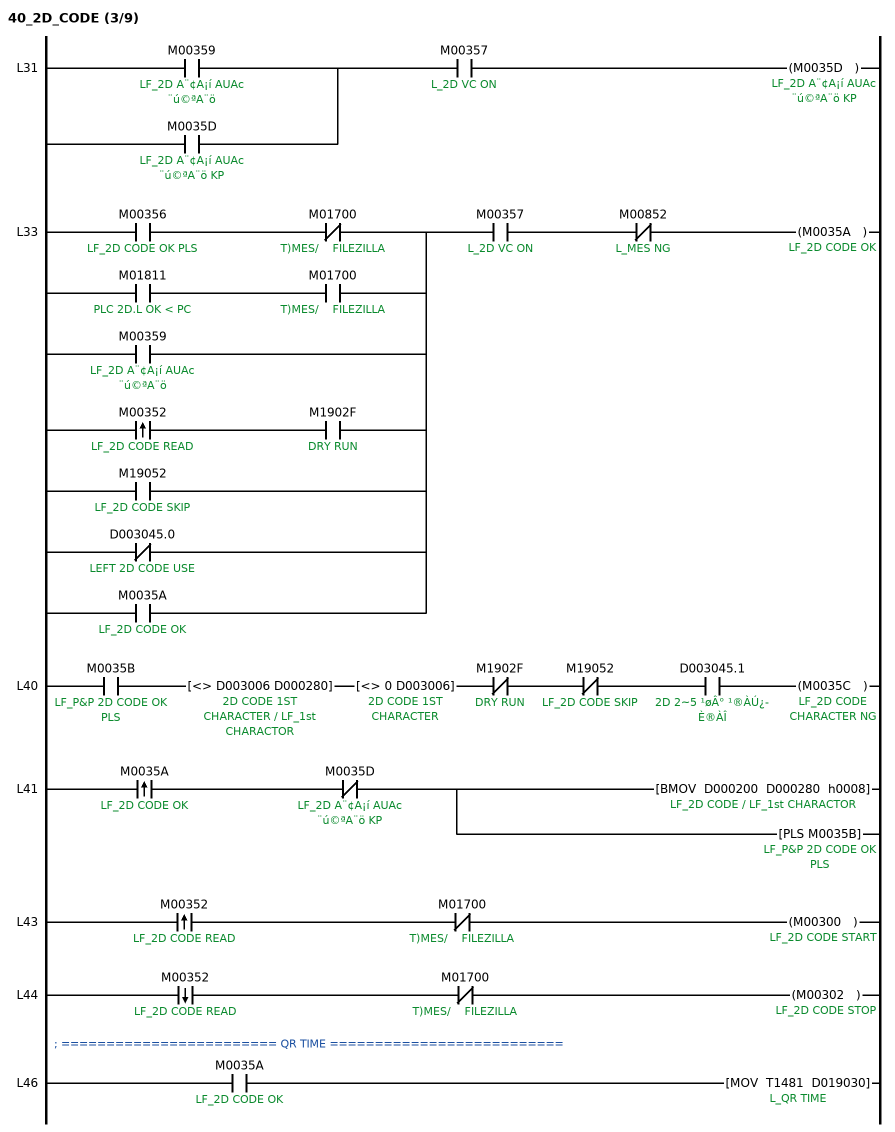
[picture p240: 40_2D_CODE rungs L31-L46]
; L31
LOAD      M00359	// LF_2D A¨¢A¡í AUAc ¨ú©ªA¨ö
OR        M0035D	// LF_2D A¨¢A¡í AUAc ¨ú©ªA¨ö KP
AND       M00357	// L_2D VC ON
OUT       M0035D	// LF_2D A¨¢A¡í AUAc ¨ú©ªA¨ö KP
; L33
LOAD      M00356	// LF_2D CODE OK PLS
AND NOT   M01700	// T)MES/    FILEZILLA
LOAD      M01811	// PLC 2D.L OK < PC
AND       M01700	// T)MES/    FILEZILLA
OR LOAD
OR        M00359	// LF_2D A¨¢A¡í AUAc ¨ú©ªA¨ö
LOADP     M00352	// LF_2D CODE READ
AND       M1902F	// DRY RUN
OR LOAD
OR        M19052	// LF_2D CODE SKIP
OR NOT    D003045.0	// LEFT 2D CODE USE
OR        M0035A	// LF_2D CODE OK
AND       M00357	// L_2D VC ON
AND NOT   M00852	// L_MES NG
OUT       M0035A	// LF_2D CODE OK
; L40
LOAD      M0035B	// LF_P&P 2D CODE OK PLS
AND<>     D003006 D000280	// 2D CODE 1ST CHARACTER / LF_1st CHARACTOR
AND<>     0 D003006	// 2D CODE 1ST CHARACTER
AND NOT   M1902F	// DRY RUN
AND NOT   M19052	// LF_2D CODE SKIP
AND       D003045.1	// 2D 2~5 ¹øÂ° ¹®ÀÚ¿­ È®ÀÎ
OUT       M0035C	// LF_2D CODE CHARACTER NG
; L41
LOADP     M0035A	// LF_2D CODE OK
AND NOT   M0035D	// LF_2D A¨¢A¡í AUAc ¨ú©ªA¨ö KP
BMOV      D000200 D000280 h0008	// LF_2D CODE / LF_1st CHARACTOR
OUTP      M0035B	// LF_P&P 2D CODE OK PLS
; L43
LOADP     M00352	// LF_2D CODE READ
AND NOT   M01700	// T)MES/    FILEZILLA
OUT       M00300	// LF_2D CODE START
; L44
LOADN     M00352	// LF_2D CODE READ
AND NOT   M01700	// T)MES/    FILEZILLA
OUT       M00302	// LF_2D CODE STOP
// ======================== QR TIME ==========================
; L46
LOAD      M0035A	// LF_2D CODE OK
MOV       T1481 D019030	// L_QR TIME

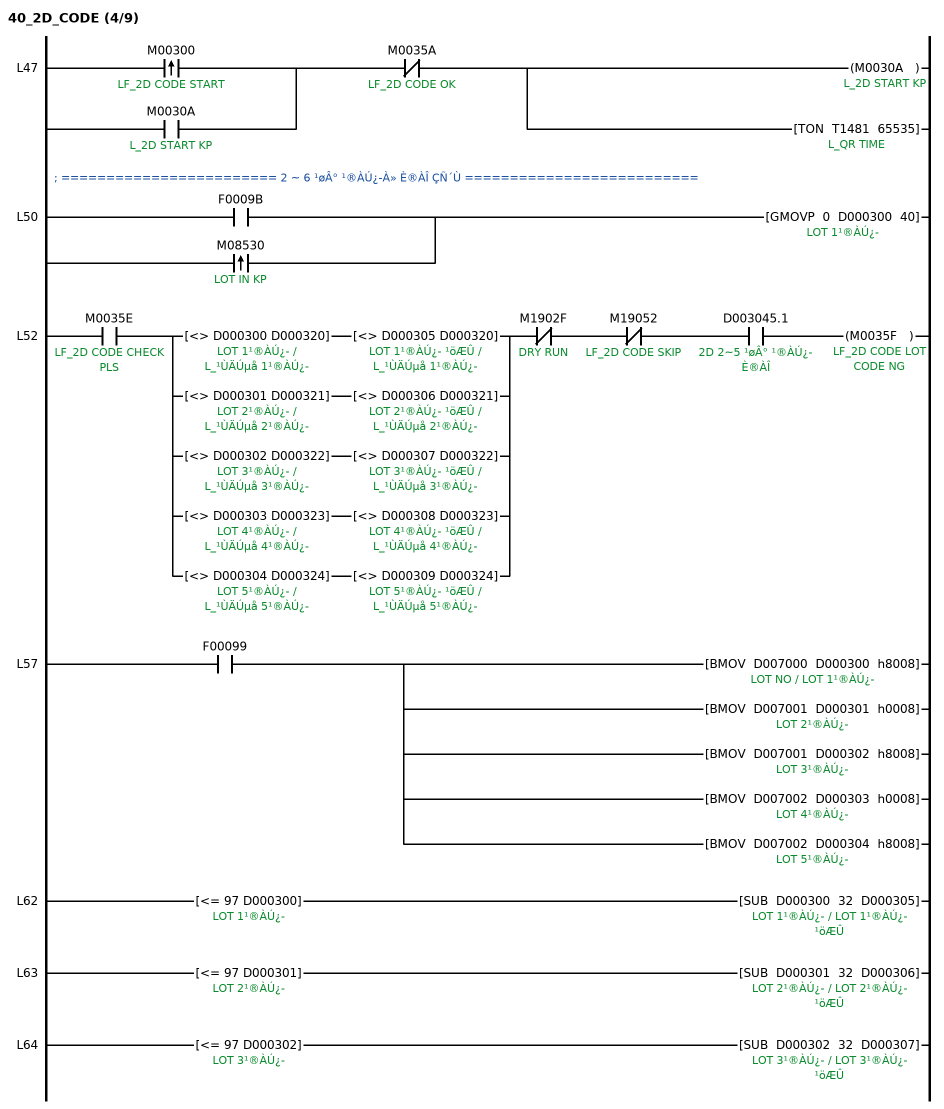
; L47
LOADP     M00300	// LF_2D CODE START
OR        M0030A	// L_2D START KP
AND NOT   M0035A	// LF_2D CODE OK
OUT       M0030A	// L_2D START KP
TON       T1481 65535	// L_QR TIME
// ======================== 2 ~ 6 ¹øÂ° ¹®ÀÚ¿­À» È®ÀÎ ÇÑ´Ù ==========================
; L50
LOAD      F0009B
ORP       M08530	// LOT IN KP
GMOVP     0 D000300 40	// LOT 1¹®ÀÚ¿­
; L52
LOAD      M0035E	// LF_2D CODE CHECK PLS
LOAD<>    D000300 D000320	// LOT 1¹®ÀÚ¿­ / L_¹ÙÄÚµå 1¹®ÀÚ¿­
AND<>     D000305 D000320	// LOT 1¹®ÀÚ¿­ ¹öÆÛ / L_¹ÙÄÚµå 1¹®ÀÚ¿­
LOAD<>    D000301 D000321	// LOT 2¹®ÀÚ¿­ / L_¹ÙÄÚµå 2¹®ÀÚ¿­
AND<>     D000306 D000321	// LOT 2¹®ÀÚ¿­ ¹öÆÛ / L_¹ÙÄÚµå 2¹®ÀÚ¿­
OR LOAD
LOAD<>    D000302 D000322	// LOT 3¹®ÀÚ¿­ / L_¹ÙÄÚµå 3¹®ÀÚ¿­
AND<>     D000307 D000322	// LOT 3¹®ÀÚ¿­ ¹öÆÛ / L_¹ÙÄÚµå 3¹®ÀÚ¿­
OR LOAD
LOAD<>    D000303 D000323	// LOT 4¹®ÀÚ¿­ / L_¹ÙÄÚµå 4¹®ÀÚ¿­
AND<>     D000308 D000323	// LOT 4¹®ÀÚ¿­ ¹öÆÛ / L_¹ÙÄÚµå 4¹®ÀÚ¿­
OR LOAD
LOAD<>    D000304 D000324	// LOT 5¹®ÀÚ¿­ / L_¹ÙÄÚµå 5¹®ÀÚ¿­
AND<>     D000309 D000324	// LOT 5¹®ÀÚ¿­ ¹öÆÛ / L_¹ÙÄÚµå 5¹®ÀÚ¿­
OR LOAD
AND LOAD
AND NOT   M1902F	// DRY RUN
AND NOT   M19052	// LF_2D CODE SKIP
AND       D003045.1	// 2D 2~5 ¹øÂ° ¹®ÀÚ¿­ È®ÀÎ
OUT       M0035F	// LF_2D CODE LOT CODE NG
; L57
LOAD      F00099
BMOV      D007000 D000300 h8008	// LOT NO / LOT 1¹®ÀÚ¿­
BMOV      D007001 D000301 h0008	// LOT 2¹®ÀÚ¿­
BMOV      D007001 D000302 h8008	// LOT 3¹®ÀÚ¿­
BMOV      D007002 D000303 h0008	// LOT 4¹®ÀÚ¿­
BMOV      D007002 D000304 h8008	// LOT 5¹®ÀÚ¿­
; L62
LOAD<=    97 D000300	// LOT 1¹®ÀÚ¿­
SUB       D000300 32 D000305	// LOT 1¹®ÀÚ¿­ / LOT 1¹®ÀÚ¿­ ¹öÆÛ
; L63
LOAD<=    97 D000301	// LOT 2¹®ÀÚ¿­
SUB       D000301 32 D000306	// LOT 2¹®ÀÚ¿­ / LOT 2¹®ÀÚ¿­ ¹öÆÛ
; L64
LOAD<=    97 D000302	// LOT 3¹®ÀÚ¿­
SUB       D000302 32 D000307	// LOT 3¹®ÀÚ¿­ / LOT 3¹®ÀÚ¿­ ¹öÆÛ

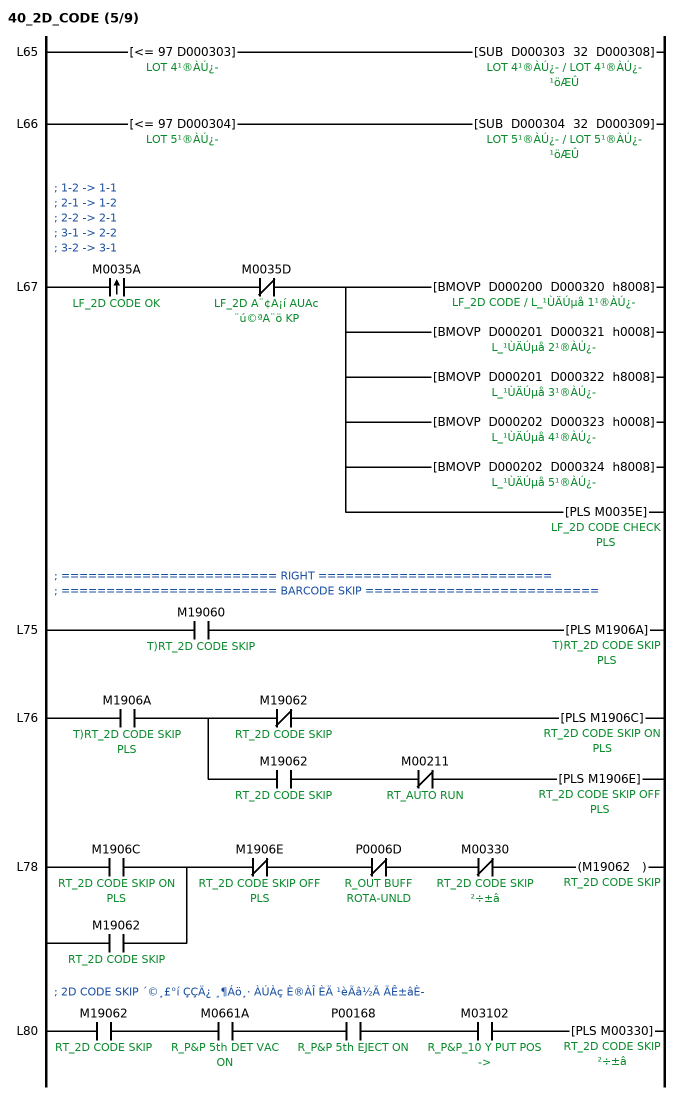
; L65
LOAD<=    97 D000303	// LOT 4¹®ÀÚ¿­
SUB       D000303 32 D000308	// LOT 4¹®ÀÚ¿­ / LOT 4¹®ÀÚ¿­ ¹öÆÛ
; L66
LOAD<=    97 D000304	// LOT 5¹®ÀÚ¿­
SUB       D000304 32 D000309	// LOT 5¹®ÀÚ¿­ / LOT 5¹®ÀÚ¿­ ¹öÆÛ
; L67
LOADP     M0035A	// LF_2D CODE OK
AND NOT   M0035D	// LF_2D A¨¢A¡í AUAc ¨ú©ªA¨ö KP
BMOVP     D000200 D000320 h8008	// LF_2D CODE / L_¹ÙÄÚµå 1¹®ÀÚ¿­
BMOVP     D000201 D000321 h0008	// L_¹ÙÄÚµå 2¹®ÀÚ¿­
BMOVP     D000201 D000322 h8008	// L_¹ÙÄÚµå 3¹®ÀÚ¿­
BMOVP     D000202 D000323 h0008	// L_¹ÙÄÚµå 4¹®ÀÚ¿­
BMOVP     D000202 D000324 h8008	// L_¹ÙÄÚµå 5¹®ÀÚ¿­
OUTP      M0035E	// LF_2D CODE CHECK PLS
// output comment: 1-2 -> 1-1
// output comment: 2-1 -> 1-2
// output comment: 2-2 -> 2-1
// output comment: 3-1 -> 2-2
// output comment: 3-2 -> 3-1
// ======================== RIGHT ==========================
// ======================== BARCODE SKIP ==========================
; L75
LOAD      M19060	// T)RT_2D CODE SKIP
OUTP      M1906A	// T)RT_2D CODE SKIP PLS
; L76
LOAD      M1906A	// T)RT_2D CODE SKIP PLS
MPUSH
AND NOT   M19062	// RT_2D CODE SKIP
OUTP      M1906C	// RT_2D CODE SKIP ON PLS
MPOP
AND       M19062	// RT_2D CODE SKIP
AND NOT   M00211	// RT_AUTO RUN
OUTP      M1906E	// RT_2D CODE SKIP OFF PLS
; L78
LOAD      M1906C	// RT_2D CODE SKIP ON PLS
OR        M19062	// RT_2D CODE SKIP
AND NOT   M1906E	// RT_2D CODE SKIP OFF PLS
AND NOT   P0006D	// R_OUT BUFF ROTA-UNLD
AND NOT   M00330	// RT_2D CODE SKIP ²÷±â
OUT       M19062	// RT_2D CODE SKIP
; L80
LOAD      M19062	// RT_2D CODE SKIP
AND       M0661A	// R_P&P 5th DET VAC ON
AND       P00168	// R_P&P 5th EJECT ON
AND       M03102	// R_P&P_10 Y PUT POS ->
OUTP      M00330	// RT_2D CODE SKIP ²÷±â
// output comment: 2D CODE SKIP ´©¸£°í ÇÇÄ¿ ¸¶Áö¸· ÀÚÀç È®ÀÎ ÈÄ ¹èÃâ½Ã ÃÊ±âÈ­

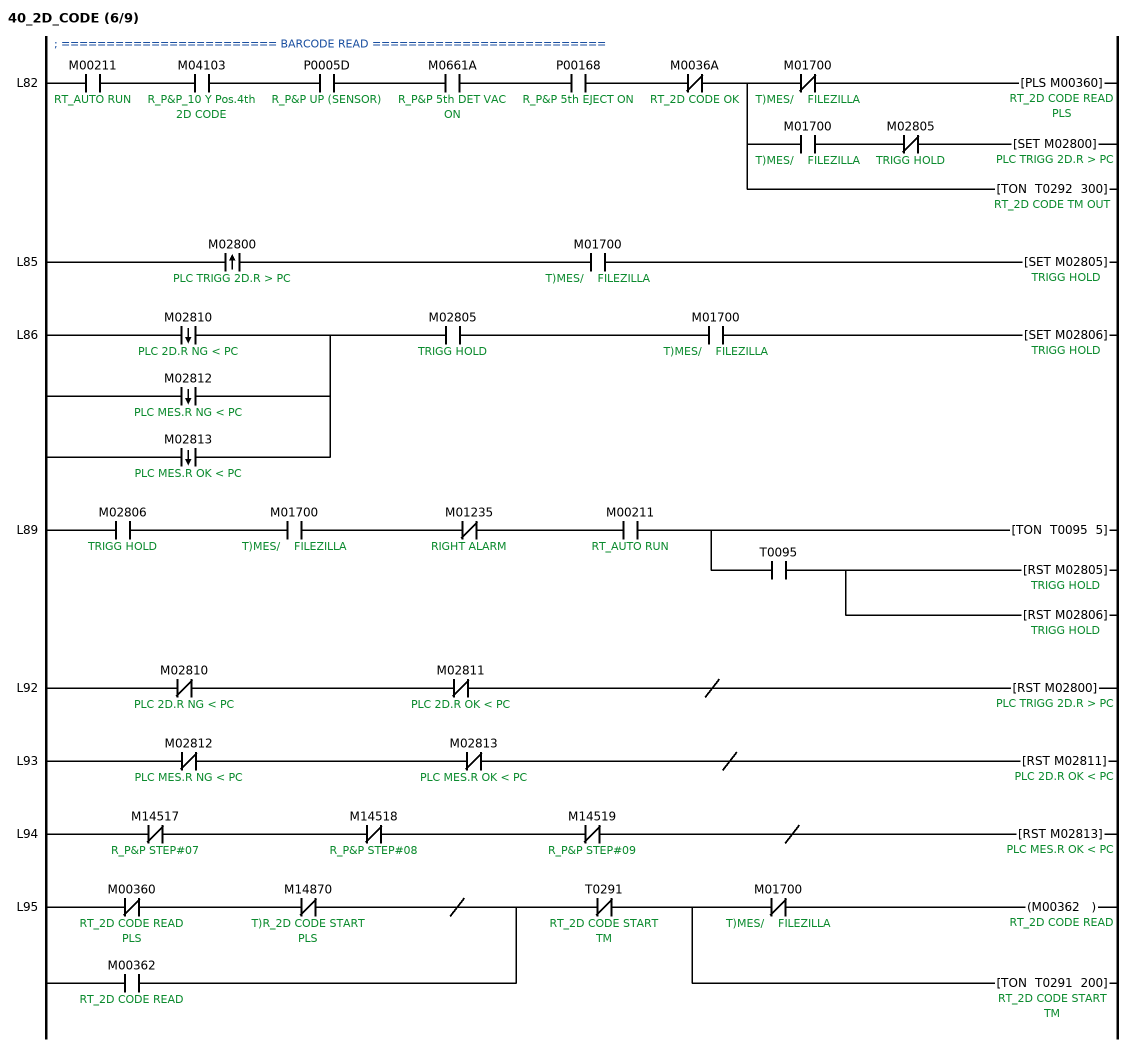
// ======================== BARCODE READ ==========================
; L82
LOAD      M00211	// RT_AUTO RUN
AND       M04103	// R_P&P_10 Y Pos.4th 2D CODE
AND       P0005D	// R_P&P UP (SENSOR)
AND       M0661A	// R_P&P 5th DET VAC ON
AND       P00168	// R_P&P 5th EJECT ON
AND NOT   M0036A	// RT_2D CODE OK
MPUSH
AND NOT   M01700	// T)MES/    FILEZILLA
OUTP      M00360	// RT_2D CODE READ PLS
MLOAD
AND       M01700	// T)MES/    FILEZILLA
AND NOT   M02805	// TRIGG HOLD
SET       M02800	// PLC TRIGG 2D.R > PC
MPOP
TON       T0292 300	// RT_2D CODE TM OUT
; L85
LOADP     M02800	// PLC TRIGG 2D.R > PC
AND       M01700	// T)MES/    FILEZILLA
SET       M02805	// TRIGG HOLD
; L86
LOADN     M02810	// PLC 2D.R NG < PC
ORN       M02812	// PLC MES.R NG < PC
ORN       M02813	// PLC MES.R OK < PC
AND       M02805	// TRIGG HOLD
AND       M01700	// T)MES/    FILEZILLA
SET       M02806	// TRIGG HOLD
; L89
LOAD      M02806	// TRIGG HOLD
AND       M01700	// T)MES/    FILEZILLA
AND NOT   M01235	// RIGHT ALARM
AND       M00211	// RT_AUTO RUN
TON       T0095 5
AND       T0095
RST       M02805	// TRIGG HOLD
RST       M02806	// TRIGG HOLD
; L92
LOAD NOT  M02810	// PLC 2D.R NG < PC
AND NOT   M02811	// PLC 2D.R OK < PC
NOT
RST       M02800	// PLC TRIGG 2D.R > PC
; L93
LOAD NOT  M02812	// PLC MES.R NG < PC
AND NOT   M02813	// PLC MES.R OK < PC
NOT
RST       M02811	// PLC 2D.R OK < PC
; L94
LOAD NOT  M14517	// R_P&P STEP#07
AND NOT   M14518	// R_P&P STEP#08
AND NOT   M14519	// R_P&P STEP#09
NOT
RST       M02813	// PLC MES.R OK < PC
; L95
LOAD NOT  M00360	// RT_2D CODE READ PLS
AND NOT   M14870	// T)R_2D CODE START PLS
NOT
OR        M00362	// RT_2D CODE READ
AND NOT   T0291	// RT_2D CODE START TM
MPUSH
AND NOT   M01700	// T)MES/    FILEZILLA
OUT       M00362	// RT_2D CODE READ
MPOP
TON       T0291 200	// RT_2D CODE START TM

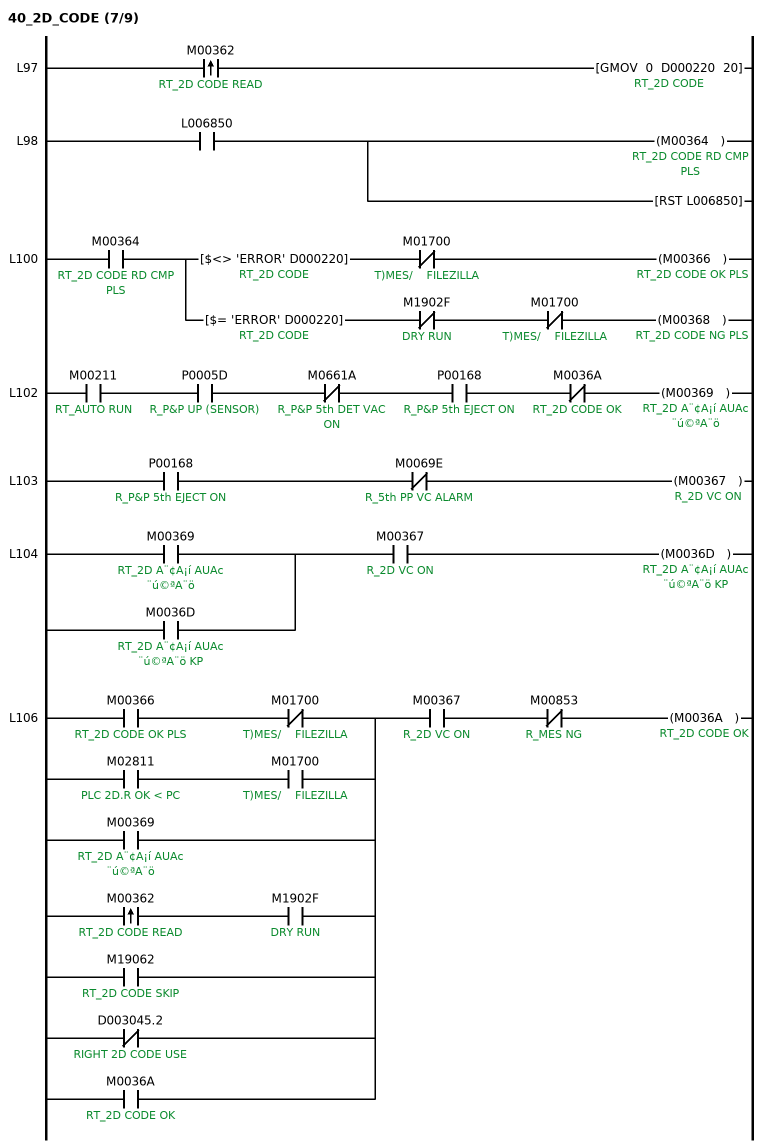
; L97
LOADP     M00362	// RT_2D CODE READ
GMOV      0 D000220 20	// RT_2D CODE
; L98
LOAD      L006850
OUT       M00364	// RT_2D CODE RD CMP PLS
RST       L006850
; L100
LOAD      M00364	// RT_2D CODE RD CMP PLS
MPUSH
AND$<>    'ERROR' D000220	// RT_2D CODE
AND NOT   M01700	// T)MES/    FILEZILLA
OUT       M00366	// RT_2D CODE OK PLS
MPOP
AND$=     'ERROR' D000220	// RT_2D CODE
AND NOT   M1902F	// DRY RUN
AND NOT   M01700	// T)MES/    FILEZILLA
OUT       M00368	// RT_2D CODE NG PLS
; L102
LOAD      M00211	// RT_AUTO RUN
AND       P0005D	// R_P&P UP (SENSOR)
AND NOT   M0661A	// R_P&P 5th DET VAC ON
AND       P00168	// R_P&P 5th EJECT ON
AND NOT   M0036A	// RT_2D CODE OK
OUT       M00369	// RT_2D A¨¢A¡í AUAc ¨ú©ªA¨ö
; L103
LOAD      P00168	// R_P&P 5th EJECT ON
AND NOT   M0069E	// R_5th PP VC ALARM
OUT       M00367	// R_2D VC ON
; L104
LOAD      M00369	// RT_2D A¨¢A¡í AUAc ¨ú©ªA¨ö
OR        M0036D	// RT_2D A¨¢A¡í AUAc ¨ú©ªA¨ö KP
AND       M00367	// R_2D VC ON
OUT       M0036D	// RT_2D A¨¢A¡í AUAc ¨ú©ªA¨ö KP
; L106
LOAD      M00366	// RT_2D CODE OK PLS
AND NOT   M01700	// T)MES/    FILEZILLA
LOAD      M02811	// PLC 2D.R OK < PC
AND       M01700	// T)MES/    FILEZILLA
OR LOAD
OR        M00369	// RT_2D A¨¢A¡í AUAc ¨ú©ªA¨ö
LOADP     M00362	// RT_2D CODE READ
AND       M1902F	// DRY RUN
OR LOAD
OR        M19062	// RT_2D CODE SKIP
OR NOT    D003045.2	// RIGHT 2D CODE USE
OR        M0036A	// RT_2D CODE OK
AND       M00367	// R_2D VC ON
AND NOT   M00853	// R_MES NG
OUT       M0036A	// RT_2D CODE OK

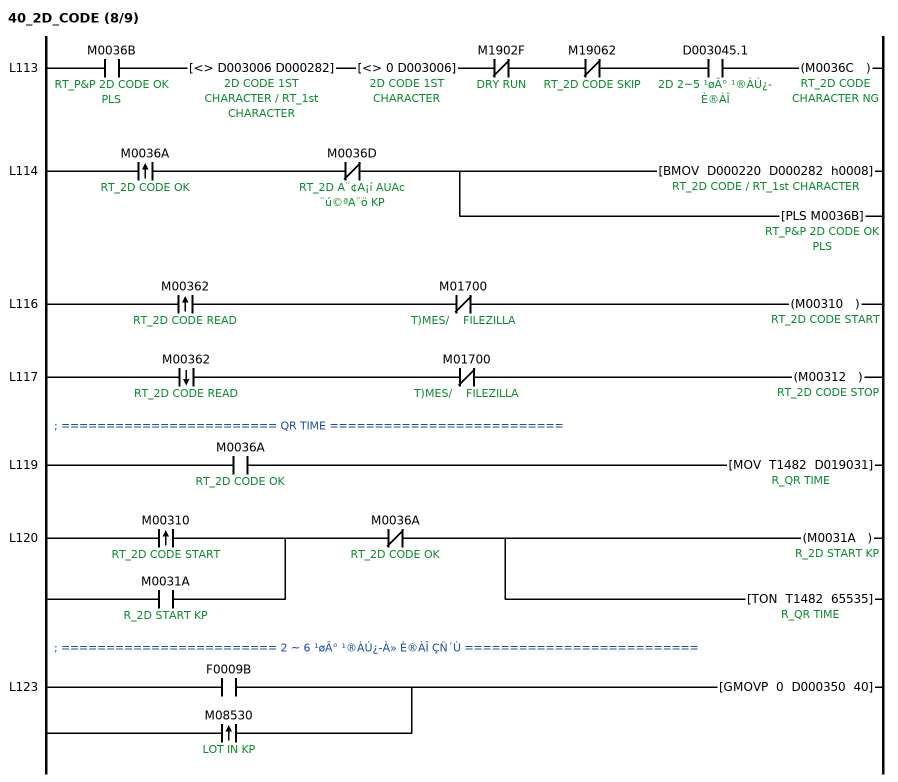
; L113
LOAD      M0036B	// RT_P&P 2D CODE OK PLS
AND<>     D003006 D000282	// 2D CODE 1ST CHARACTER / RT_1st CHARACTER
AND<>     0 D003006	// 2D CODE 1ST CHARACTER
AND NOT   M1902F	// DRY RUN
AND NOT   M19062	// RT_2D CODE SKIP
AND       D003045.1	// 2D 2~5 ¹øÂ° ¹®ÀÚ¿­ È®ÀÎ
OUT       M0036C	// RT_2D CODE CHARACTER NG
; L114
LOADP     M0036A	// RT_2D CODE OK
AND NOT   M0036D	// RT_2D A¨¢A¡í AUAc ¨ú©ªA¨ö KP
BMOV      D000220 D000282 h0008	// RT_2D CODE / RT_1st CHARACTER
OUTP      M0036B	// RT_P&P 2D CODE OK PLS
; L116
LOADP     M00362	// RT_2D CODE READ
AND NOT   M01700	// T)MES/    FILEZILLA
OUT       M00310	// RT_2D CODE START
; L117
LOADN     M00362	// RT_2D CODE READ
AND NOT   M01700	// T)MES/    FILEZILLA
OUT       M00312	// RT_2D CODE STOP
// ======================== QR TIME ==========================
; L119
LOAD      M0036A	// RT_2D CODE OK
MOV       T1482 D019031	// R_QR TIME
; L120
LOADP     M00310	// RT_2D CODE START
OR        M0031A	// R_2D START KP
AND NOT   M0036A	// RT_2D CODE OK
OUT       M0031A	// R_2D START KP
TON       T1482 65535	// R_QR TIME
// ======================== 2 ~ 6 ¹øÂ° ¹®ÀÚ¿­À» È®ÀÎ ÇÑ´Ù ==========================
; L123
LOAD      F0009B
ORP       M08530	// LOT IN KP
GMOVP     0 D000350 40

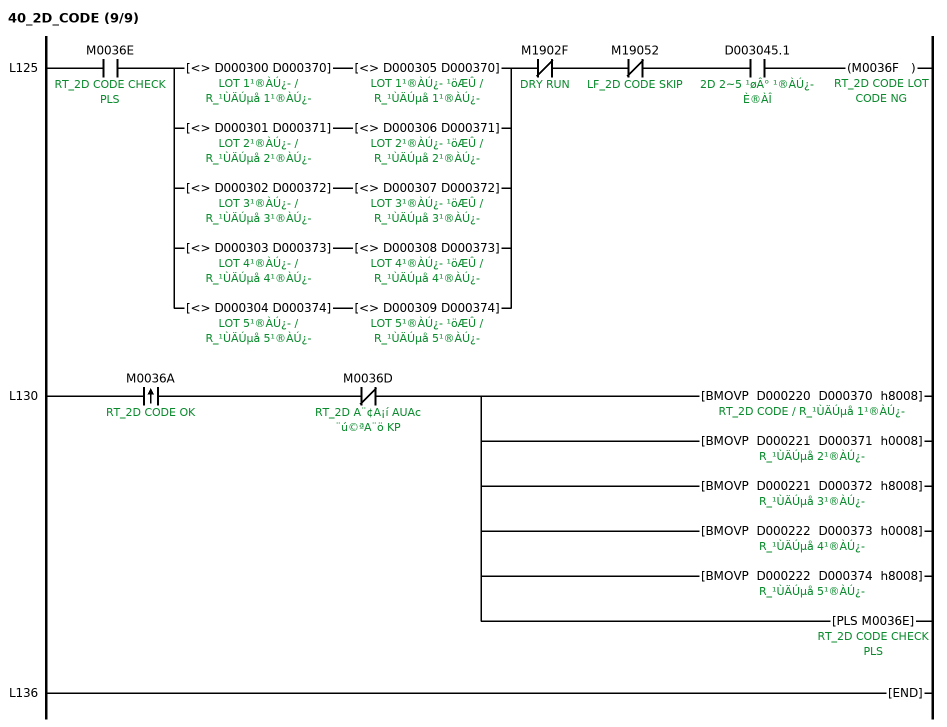
; L125
LOAD      M0036E	// RT_2D CODE CHECK PLS
LOAD<>    D000300 D000370	// LOT 1¹®ÀÚ¿­ / R_¹ÙÄÚµå 1¹®ÀÚ¿­
AND<>     D000305 D000370	// LOT 1¹®ÀÚ¿­ ¹öÆÛ / R_¹ÙÄÚµå 1¹®ÀÚ¿­
LOAD<>    D000301 D000371	// LOT 2¹®ÀÚ¿­ / R_¹ÙÄÚµå 2¹®ÀÚ¿­
AND<>     D000306 D000371	// LOT 2¹®ÀÚ¿­ ¹öÆÛ / R_¹ÙÄÚµå 2¹®ÀÚ¿­
OR LOAD
LOAD<>    D000302 D000372	// LOT 3¹®ÀÚ¿­ / R_¹ÙÄÚµå 3¹®ÀÚ¿­
AND<>     D000307 D000372	// LOT 3¹®ÀÚ¿­ ¹öÆÛ / R_¹ÙÄÚµå 3¹®ÀÚ¿­
OR LOAD
LOAD<>    D000303 D000373	// LOT 4¹®ÀÚ¿­ / R_¹ÙÄÚµå 4¹®ÀÚ¿­
AND<>     D000308 D000373	// LOT 4¹®ÀÚ¿­ ¹öÆÛ / R_¹ÙÄÚµå 4¹®ÀÚ¿­
OR LOAD
LOAD<>    D000304 D000374	// LOT 5¹®ÀÚ¿­ / R_¹ÙÄÚµå 5¹®ÀÚ¿­
AND<>     D000309 D000374	// LOT 5¹®ÀÚ¿­ ¹öÆÛ / R_¹ÙÄÚµå 5¹®ÀÚ¿­
OR LOAD
AND LOAD
AND NOT   M1902F	// DRY RUN
AND NOT   M19052	// LF_2D CODE SKIP
AND       D003045.1	// 2D 2~5 ¹øÂ° ¹®ÀÚ¿­ È®ÀÎ
OUT       M0036F	// RT_2D CODE LOT CODE NG
; L130
LOADP     M0036A	// RT_2D CODE OK
AND NOT   M0036D	// RT_2D A¨¢A¡í AUAc ¨ú©ªA¨ö KP
BMOVP     D000220 D000370 h8008	// RT_2D CODE / R_¹ÙÄÚµå 1¹®ÀÚ¿­
BMOVP     D000221 D000371 h0008	// R_¹ÙÄÚµå 2¹®ÀÚ¿­
BMOVP     D000221 D000372 h8008	// R_¹ÙÄÚµå 3¹®ÀÚ¿­
BMOVP     D000222 D000373 h0008	// R_¹ÙÄÚµå 4¹®ÀÚ¿­
BMOVP     D000222 D000374 h8008	// R_¹ÙÄÚµå 5¹®ÀÚ¿­
OUTP      M0036E	// RT_2D CODE CHECK PLS
; L136
END

PROGRAM 41_MES (task: ½ºÄµ ÇÁ·Î±×·¥)

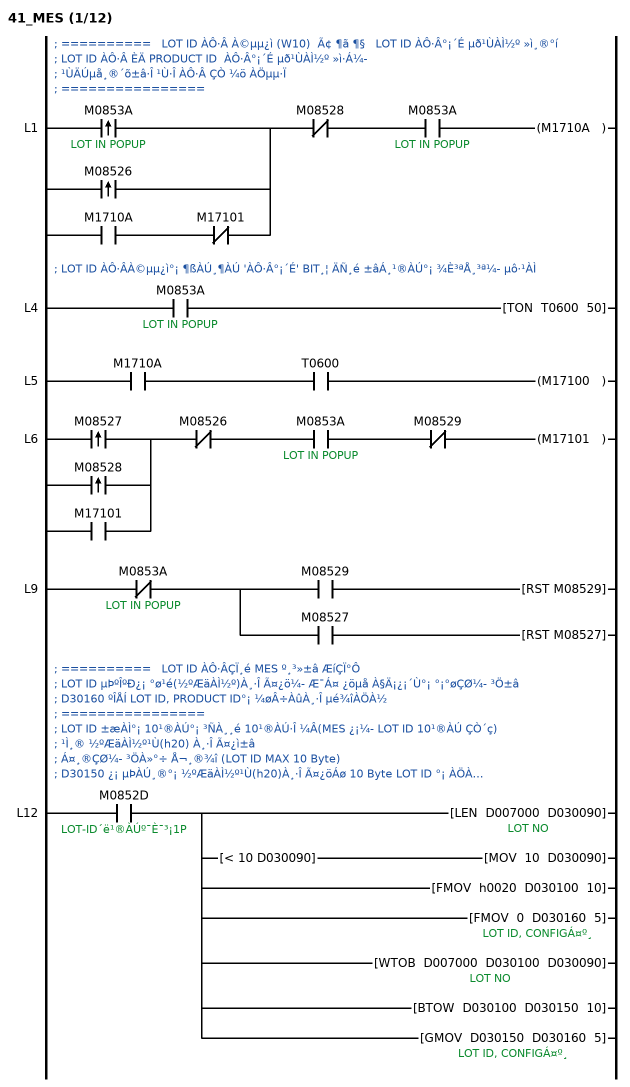
// ==========   LOT ID ÀÔ·Â À©µµ¿ì (W10)  Ã¢ ¶ã ¶§   LOT ID ÀÔ·Â°¡´É µð¹ÙÀÌ½º »ì¸®°í
//    LOT ID ÀÔ·Â ÈÄ PRODUCT ID  ÀÔ·Â°¡´É µð¹ÙÀÌ½º »ì·Á¼­ 
//    ¹ÙÄÚµå¸®´õ±â·Î ¹Ù·Î ÀÔ·Â ÇÒ ¼ö ÀÖµµ·Ï
// ================
; L1
LOADP     M0853A	// LOT IN POPUP
ORP       M08526
LOAD      M1710A
AND NOT   M17101
OR LOAD
AND NOT   M08528
AND       M0853A	// LOT IN POPUP
OUT       M1710A
; L4
LOAD      M0853A	// LOT IN POPUP
TON       T0600 50
// output comment: LOT ID ÀÔ·ÂÀ©µµ¿ì°¡ ¶ßÀÚ¸¶ÀÚ 'ÀÔ·Â°¡´É' BIT¸¦ ÄÑ¸é ±âÁ¸¹®ÀÚ°¡ ¾È³ªÅ¸³ª¼­ µô·¹ÀÌ
; L5
LOAD      M1710A
AND       T0600
OUT       M17100
; L6
LOADP     M08527
ORP       M08528
OR        M17101
AND NOT   M08526
AND       M0853A	// LOT IN POPUP
AND NOT   M08529
OUT       M17101
; L9
LOAD NOT  M0853A	// LOT IN POPUP
MPUSH
AND       M08529
RST       M08529
MPOP
AND       M08527
RST       M08527
// ==========   LOT ID ÀÔ·ÂÇÏ¸é MES º¸³»±â ÆíÇÏ°Ô
//    LOT ID µÞºÎºÐ¿¡ °ø¹é(½ºÆäÀÌ½º)À¸·Î Ã¤¿ö¼­ Æ¯Á¤ ¿öµå À§Ä¡¿¡´Ù°¡ °¡°øÇØ¼­ ³Ö±â
//   D30160 ºÎÅÍ LOT ID, PRODUCT ID°¡ ¼øÂ÷ÀûÀ¸·Î µé¾îÀÖÀ½
// ================
; L12
LOAD      M0852D	// LOT-ID´ë¹®ÀÚº¯È¯³¡1P
LEN       D007000 D030090	// LOT NO
MPUSH
AND<      10 D030090
MOV       10 D030090
MPOP
FMOV      h0020 D030100 10
FMOV      0 D030160 5	// LOT ID, CONFIGÁ¤º¸
WTOB      D007000 D030100 D030090	// LOT NO
BTOW      D030100 D030150 10
GMOV      D030150 D030160 5	// LOT ID, CONFIGÁ¤º¸
// output comment: LOT ID ±æÀÌ°¡ 10¹®ÀÚ°¡ ³ÑÀ¸¸é 10¹®ÀÚ·Î ¼Â(MES ¿¡¼­ LOT ID 10¹®ÀÚ ÇÒ´ç)
// output comment: ¹Ì¸® ½ºÆäÀÌ½º¹Ù(h20) À¸·Î Ã¤¿ì±â
// output comment: Á¤¸®ÇØ¼­ ³ÖÀ»°÷ Å¬¸®¾î (LOT ID MAX 10 Byte)
// output comment: D30150 ¿¡ µÞÀÚ¸®°¡ ½ºÆäÀÌ½º¹Ù(h20)À¸·Î Ã¤¿öÁø 10 Byte LOT ID °¡ ÀÖÀ½
// output comment: LOT ID µé¾îÀÖ´Â ¾ÕÂÊ 5°³¿öµå (10 Byte)¸¸ ÀÌµ¿

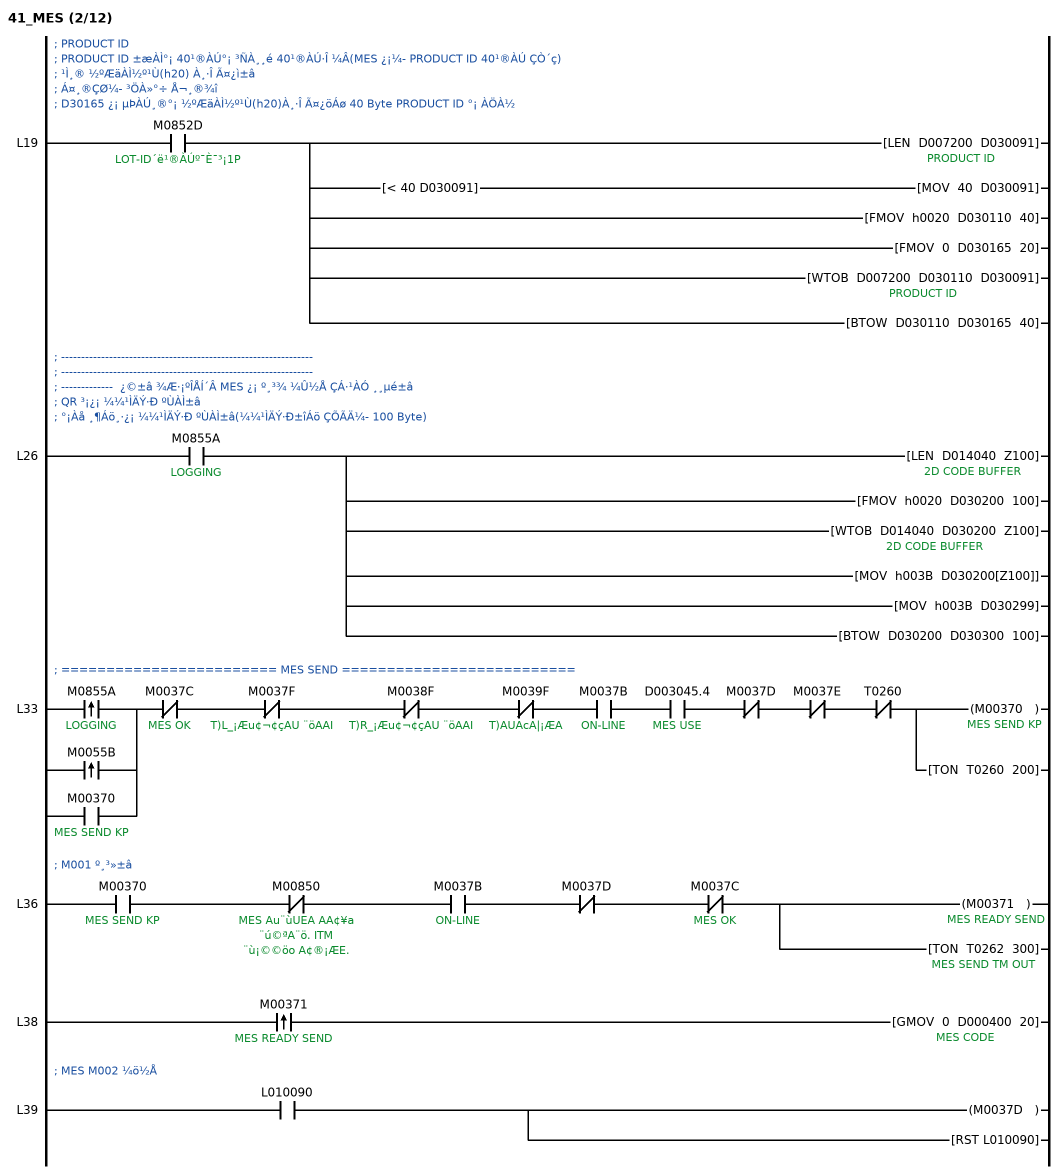
; L19
LOAD      M0852D	// LOT-ID´ë¹®ÀÚº¯È¯³¡1P
LEN       D007200 D030091	// PRODUCT ID
MPUSH
AND<      40 D030091
MOV       40 D030091
MPOP
FMOV      h0020 D030110 40
FMOV      0 D030165 20
WTOB      D007200 D030110 D030091	// PRODUCT ID
BTOW      D030110 D030165 40
// output comment: PRODUCT ID
// output comment: PRODUCT ID ±æÀÌ°¡ 40¹®ÀÚ°¡ ³ÑÀ¸¸é 40¹®ÀÚ·Î ¼Â(MES ¿¡¼­ PRODUCT ID 40¹®ÀÚ ÇÒ´ç)
// output comment: ¹Ì¸® ½ºÆäÀÌ½º¹Ù(h20) À¸·Î Ã¤¿ì±â
// output comment: Á¤¸®ÇØ¼­ ³ÖÀ»°÷ Å¬¸®¾î
// output comment: D30165 ¿¡ µÞÀÚ¸®°¡ ½ºÆäÀÌ½º¹Ù(h20)À¸·Î Ã¤¿öÁø 40 Byte PRODUCT ID °¡ ÀÖÀ½
// ---------------------------------------------------------------
// ---------------------------------------------------------------
// -------------  ¿©±â ¾Æ·¡ºÎÅÍ´Â MES ¿¡ º¸³¾ ¼Û½Å ÇÁ·¹ÀÓ ¸¸µé±â
; L26
LOAD      M0855A	// LOGGING
LEN       D014040 Z100	// 2D CODE BUFFER
FMOV      h0020 D030200 100
WTOB      D014040 D030200 Z100	// 2D CODE BUFFER
MOV       h003B D030200[Z100]
MOV       h003B D030299
BTOW      D030200 D030300 100
// output comment: QR ³¡¿¡ ¼¼¹ÌÄÝ·Ð ºÙÀÌ±â
// output comment: °¡Àå ¸¶Áö¸·¿¡ ¼¼¹ÌÄÝ·Ð ºÙÀÌ±â(¼¼¹ÌÄÝ·Ð±îÁö ÇÕÃÄ¼­ 100 Byte)
// ======================== MES SEND ==========================
; L33
LOADP     M0855A	// LOGGING
ORP       M0055B
OR        M00370	// MES SEND KP
AND NOT   M0037C	// MES OK
AND NOT   M0037F	// T)L_¡Æu¢¬¢çAU ¨öAAI
AND NOT   M0038F	// T)R_¡Æu¢¬¢çAU ¨öAAI
AND NOT   M0039F	// T)AUAcA|¡ÆA
AND       M0037B	// ON-LINE
AND       D003045.4	// MES USE
AND NOT   M0037D
AND NOT   M0037E
AND NOT   T0260
OUT       M00370	// MES SEND KP
TON       T0260 200
; L36
LOAD      M00370	// MES SEND KP
AND NOT   M00850	// MES Au¨ùUEA AA¢¥a ¨ú©ªA¨ö. ITM ¨ù¡©©öo A¢®¡ÆE.
AND       M0037B	// ON-LINE
AND NOT   M0037D
AND NOT   M0037C	// MES OK
OUT       M00371	// MES READY SEND
TON       T0262 300	// MES SEND TM OUT
// output comment: M001 º¸³»±â
; L38
LOADP     M00371	// MES READY SEND
GMOV      0 D000400 20	// MES CODE
; L39
LOAD      L010090
OUT       M0037D
RST       L010090
// output comment: MES M002 ¼ö½Å

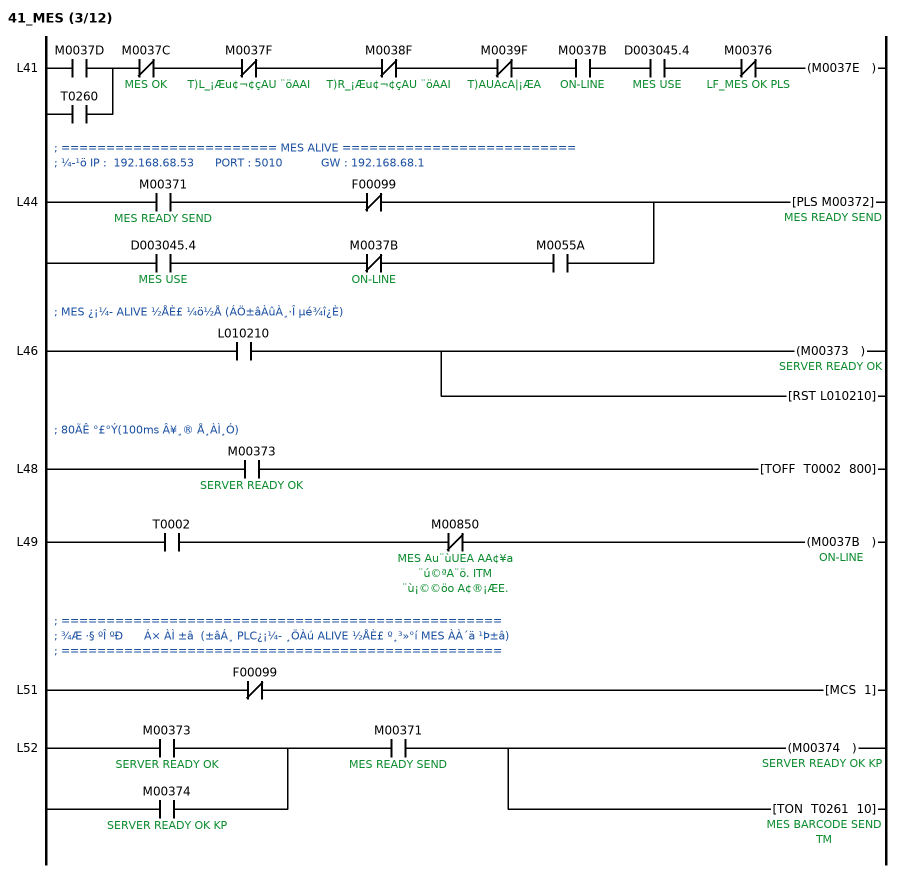
; L41
LOAD      M0037D
OR        T0260
AND NOT   M0037C	// MES OK
AND NOT   M0037F	// T)L_¡Æu¢¬¢çAU ¨öAAI
AND NOT   M0038F	// T)R_¡Æu¢¬¢çAU ¨öAAI
AND NOT   M0039F	// T)AUAcA|¡ÆA
AND       M0037B	// ON-LINE
AND       D003045.4	// MES USE
AND NOT   M00376	// LF_MES OK PLS
OUT       M0037E
// ======================== MES ALIVE ==========================
// 
// ¼­¹ö IP :  192.168.68.53      PORT : 5010           GW : 192.168.68.1
; L44
LOAD      M00371	// MES READY SEND
AND NOT   F00099
LOAD      D003045.4	// MES USE
AND NOT   M0037B	// ON-LINE
AND       M0055A
OR LOAD
OUTP      M00372	// MES READY SEND
; L46
LOAD      L010210
OUT       M00373	// SERVER READY OK
RST       L010210
// output comment: MES ¿¡¼­ ALIVE ½ÅÈ£ ¼ö½Å (ÁÖ±âÀûÀ¸·Î µé¾î¿È)
; L48
LOAD      M00373	// SERVER READY OK
TOFF      T0002 800
// output comment: 80ÃÊ °£°Ý(100ms Â¥¸® Å¸ÀÌ¸Ó)
; L49
LOAD      T0002
AND NOT   M00850	// MES Au¨ùUEA AA¢¥a ¨ú©ªA¨ö. ITM ¨ù¡©©öo A¢®¡ÆE.
OUT       M0037B	// ON-LINE
// =================================================
// 
//     ¾Æ ·§ ºÎ ºÐ      Á× ÀÌ ±â  (±âÁ¸ PLC¿¡¼­ ¸ÕÀú ALIVE ½ÅÈ£ º¸³»°í MES ÀÀ´ä ¹Þ±â)
// 
// =================================================
; L51
LOAD NOT  F00099
MCS       1
; L52
LOAD      M00373	// SERVER READY OK
OR        M00374	// SERVER READY OK KP
AND       M00371	// MES READY SEND
OUT       M00374	// SERVER READY OK KP
TON       T0261 10	// MES BARCODE SEND TM

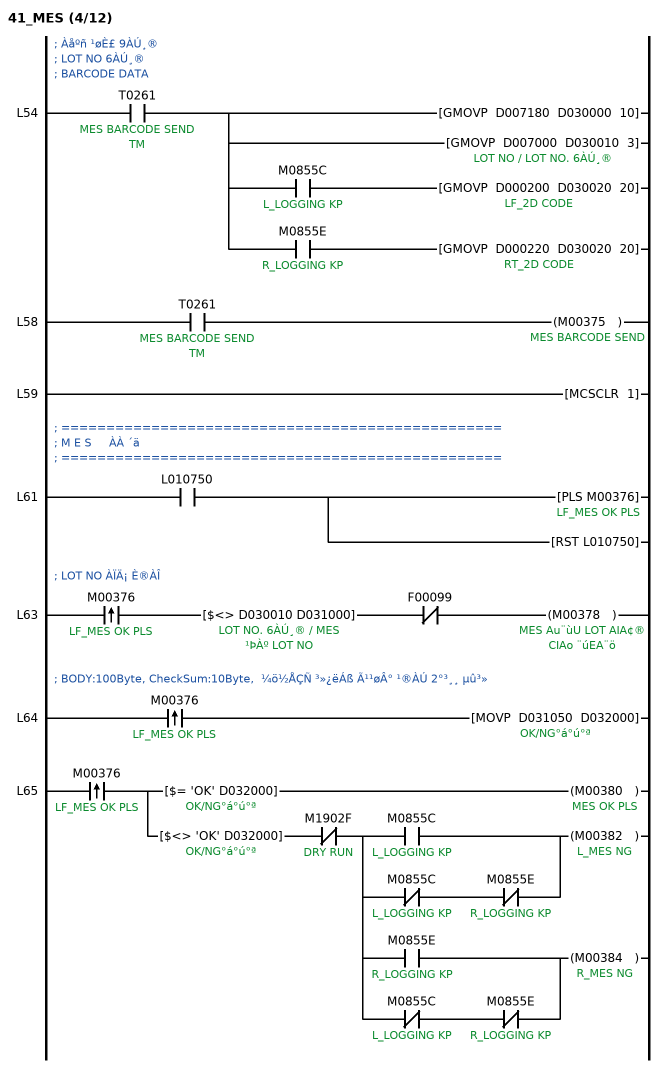
; L54
LOAD      T0261	// MES BARCODE SEND TM
GMOVP     D007180 D030000 10
GMOVP     D007000 D030010 3	// LOT NO / LOT NO. 6ÀÚ¸®
MPUSH
AND       M0855C	// L_LOGGING KP
GMOVP     D000200 D030020 20	// LF_2D CODE
MPOP
AND       M0855E	// R_LOGGING KP
GMOVP     D000220 D030020 20	// RT_2D CODE
// output comment: Àåºñ ¹øÈ£ 9ÀÚ¸®
// output comment: LOT NO 6ÀÚ¸®
// output comment: BARCODE DATA
; L58
LOAD      T0261	// MES BARCODE SEND TM
OUT       M00375	// MES BARCODE SEND
; L59
MCSCLR    1
// =================================================
// 
//    M E S     ÀÀ ´ä
// 
// =================================================
; L61
LOAD      L010750
OUTP      M00376	// LF_MES OK PLS
RST       L010750
; L63
LOADP     M00376	// LF_MES OK PLS
AND$<>    D030010 D031000	// LOT NO. 6ÀÚ¸® / MES ¹ÞÀº LOT NO
AND NOT   F00099
OUT       M00378	// MES Au¨ùU LOT AIA¢® CIAo ¨úEA¨ö
// output comment: LOT NO ÀÏÄ¡ È®ÀÎ
; L64
LOADP     M00376	// LF_MES OK PLS
MOVP      D031050 D032000	// OK/NG°á°ú°ª
// output comment: BODY:100Byte, CheckSum:10Byte,  ¼ö½ÅÇÑ ³»¿ëÁß Ã¹¹øÂ° ¹®ÀÚ 2°³¸¸ µû³»
; L65
LOADP     M00376	// LF_MES OK PLS
MPUSH
AND$=     'OK' D032000	// OK/NG°á°ú°ª
OUT       M00380	// MES OK PLS
MPOP
AND$<>    'OK' D032000	// OK/NG°á°ú°ª
AND NOT   M1902F	// DRY RUN
MPUSH
LOAD      M0855C	// L_LOGGING KP
LOAD NOT  M0855C	// L_LOGGING KP
AND NOT   M0855E	// R_LOGGING KP
OR LOAD
AND LOAD
OUT       M00382	// L_MES NG
MPOP
LOAD      M0855E	// R_LOGGING KP
LOAD NOT  M0855C	// L_LOGGING KP
AND NOT   M0855E	// R_LOGGING KP
OR LOAD
AND LOAD
OUT       M00384	// R_MES NG

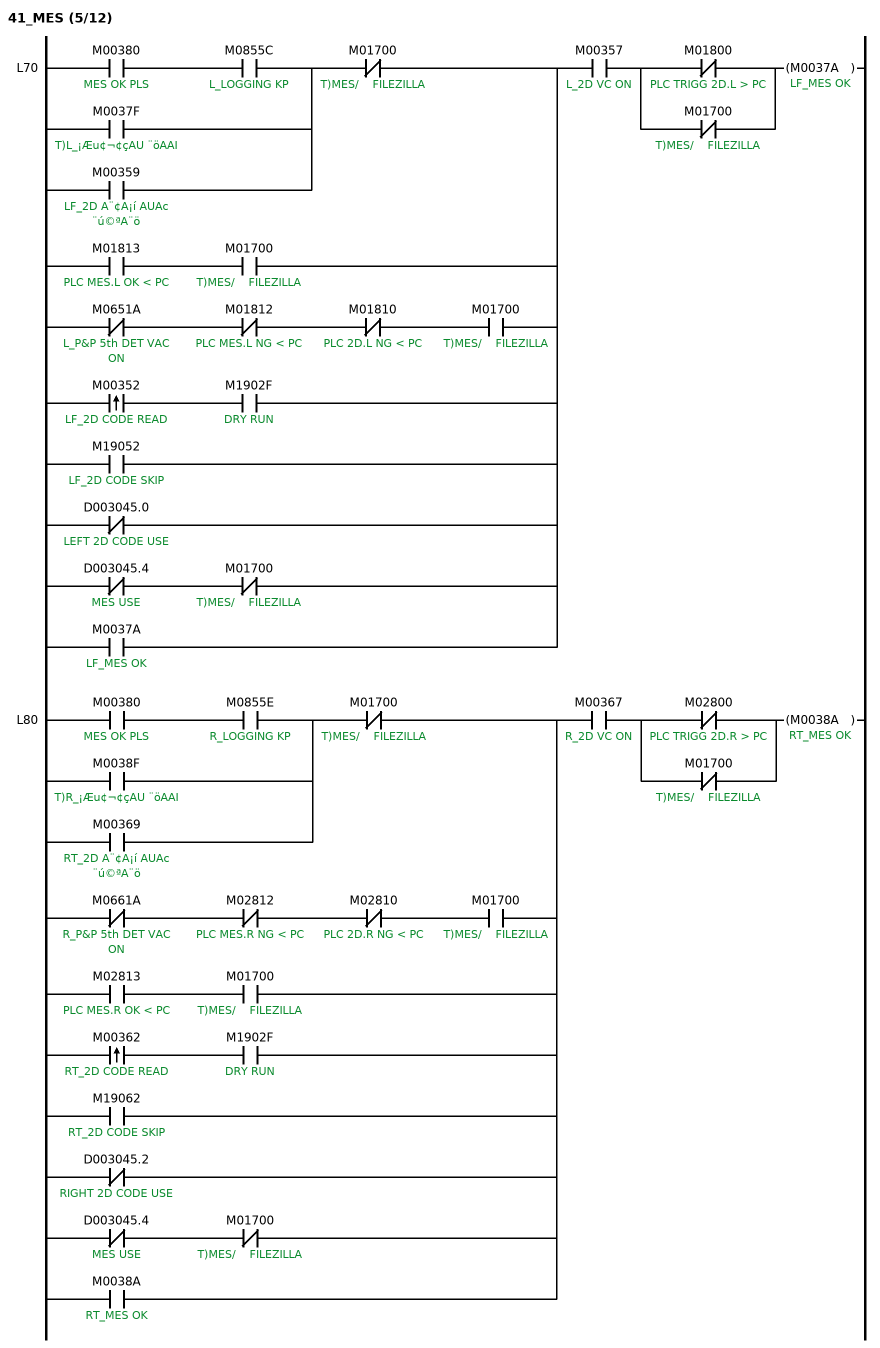
; L70
LOAD      M00380	// MES OK PLS
AND       M0855C	// L_LOGGING KP
OR        M0037F	// T)L_¡Æu¢¬¢çAU ¨öAAI
OR        M00359	// LF_2D A¨¢A¡í AUAc ¨ú©ªA¨ö
AND NOT   M01700	// T)MES/    FILEZILLA
LOAD      M01813	// PLC MES.L OK < PC
AND       M01700	// T)MES/    FILEZILLA
OR LOAD
LOAD NOT  M0651A	// L_P&P 5th DET VAC ON
AND NOT   M01812	// PLC MES.L NG < PC
AND NOT   M01810	// PLC 2D.L NG < PC
AND       M01700	// T)MES/    FILEZILLA
OR LOAD
LOADP     M00352	// LF_2D CODE READ
AND       M1902F	// DRY RUN
OR LOAD
OR        M19052	// LF_2D CODE SKIP
OR NOT    D003045.0	// LEFT 2D CODE USE
LOAD NOT  D003045.4	// MES USE
AND NOT   M01700	// T)MES/    FILEZILLA
OR LOAD
OR        M0037A	// LF_MES OK
AND       M00357	// L_2D VC ON
LOAD NOT  M01800	// PLC TRIGG 2D.L > PC
OR NOT    M01700	// T)MES/    FILEZILLA
AND LOAD
OUT       M0037A	// LF_MES OK
; L80
LOAD      M00380	// MES OK PLS
AND       M0855E	// R_LOGGING KP
OR        M0038F	// T)R_¡Æu¢¬¢çAU ¨öAAI
OR        M00369	// RT_2D A¨¢A¡í AUAc ¨ú©ªA¨ö
AND NOT   M01700	// T)MES/    FILEZILLA
LOAD NOT  M0661A	// R_P&P 5th DET VAC ON
AND NOT   M02812	// PLC MES.R NG < PC
AND NOT   M02810	// PLC 2D.R NG < PC
AND       M01700	// T)MES/    FILEZILLA
OR LOAD
LOAD      M02813	// PLC MES.R OK < PC
AND       M01700	// T)MES/    FILEZILLA
OR LOAD
LOADP     M00362	// RT_2D CODE READ
AND       M1902F	// DRY RUN
OR LOAD
OR        M19062	// RT_2D CODE SKIP
OR NOT    D003045.2	// RIGHT 2D CODE USE
LOAD NOT  D003045.4	// MES USE
AND NOT   M01700	// T)MES/    FILEZILLA
OR LOAD
OR        M0038A	// RT_MES OK
AND       M00367	// R_2D VC ON
LOAD NOT  M02800	// PLC TRIGG 2D.R > PC
OR NOT    M01700	// T)MES/    FILEZILLA
AND LOAD
OUT       M0038A	// RT_MES OK

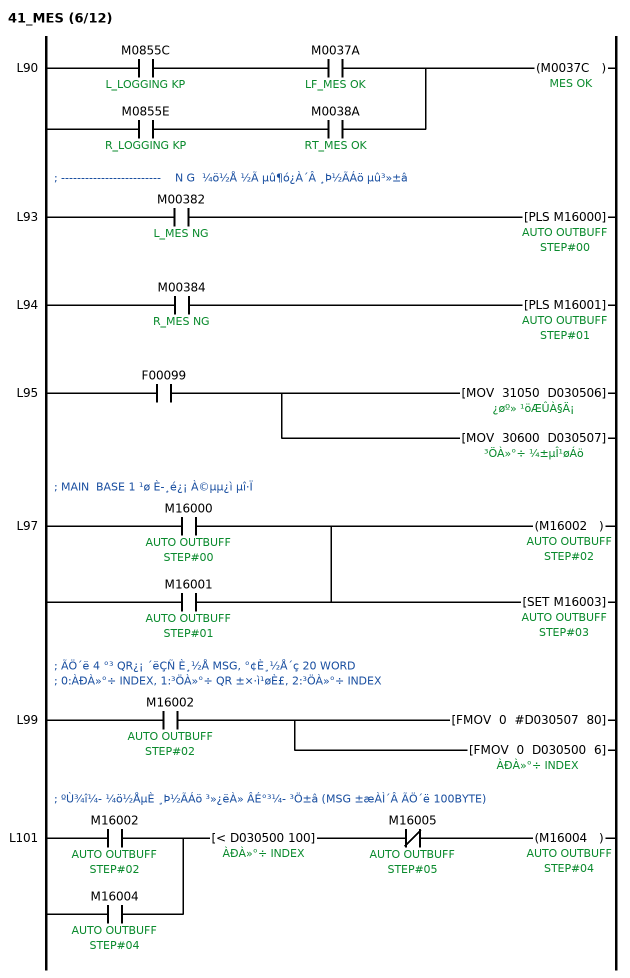
; L90
LOAD      M0855C	// L_LOGGING KP
AND       M0037A	// LF_MES OK
LOAD      M0855E	// R_LOGGING KP
AND       M0038A	// RT_MES OK
OR LOAD
OUT       M0037C	// MES OK
// -------------------------    N G  ¼ö½Å ½Ã µû¶ó¿À´Â ¸Þ½ÃÁö µû³»±â
; L93
LOAD      M00382	// L_MES NG
OUTP      M16000	// AUTO OUTBUFF STEP#00
; L94
LOAD      M00384	// R_MES NG
OUTP      M16001	// AUTO OUTBUFF STEP#01
; L95
LOAD      F00099
MOV       31050 D030506	// ¿øº» ¹öÆÛÀ§Ä¡
MOV       30600 D030507	// ³ÖÀ»°÷ ¼±µÎ¹øÁö
; L97
LOAD      M16000	// AUTO OUTBUFF STEP#00
OR        M16001	// AUTO OUTBUFF STEP#01
OUT       M16002	// AUTO OUTBUFF STEP#02
SET       M16003	// AUTO OUTBUFF STEP#03
// output comment: MAIN  BASE 1 ¹ø È­¸é¿¡ À©µµ¿ì µî·Ï
; L99
LOAD      M16002	// AUTO OUTBUFF STEP#02
FMOV      0 #D030507 80
FMOV      0 D030500 6	// ÀÐÀ»°÷ INDEX
// output comment: ÃÖ´ë 4 °³ QR¿¡ ´ëÇÑ È¸½Å MSG, °¢È¸½Å´ç 20 WORD
// output comment: 0:ÀÐÀ»°÷ INDEX, 1:³ÖÀ»°÷ QR ±×·ì¹øÈ£, 2:³ÖÀ»°÷ INDEX
; L101
LOAD      M16002	// AUTO OUTBUFF STEP#02
OR        M16004	// AUTO OUTBUFF STEP#04
AND<      D030500 100	// ÀÐÀ»°÷ INDEX
AND NOT   M16005	// AUTO OUTBUFF STEP#05
OUT       M16004	// AUTO OUTBUFF STEP#04
// output comment: ºÙ¾î¼­ ¼ö½ÅµÈ ¸Þ½ÃÁö ³»¿ëÀ» ÂÉ°³¼­ ³Ö±â (MSG ±æÀÌ´Â ÃÖ´ë 100BYTE)

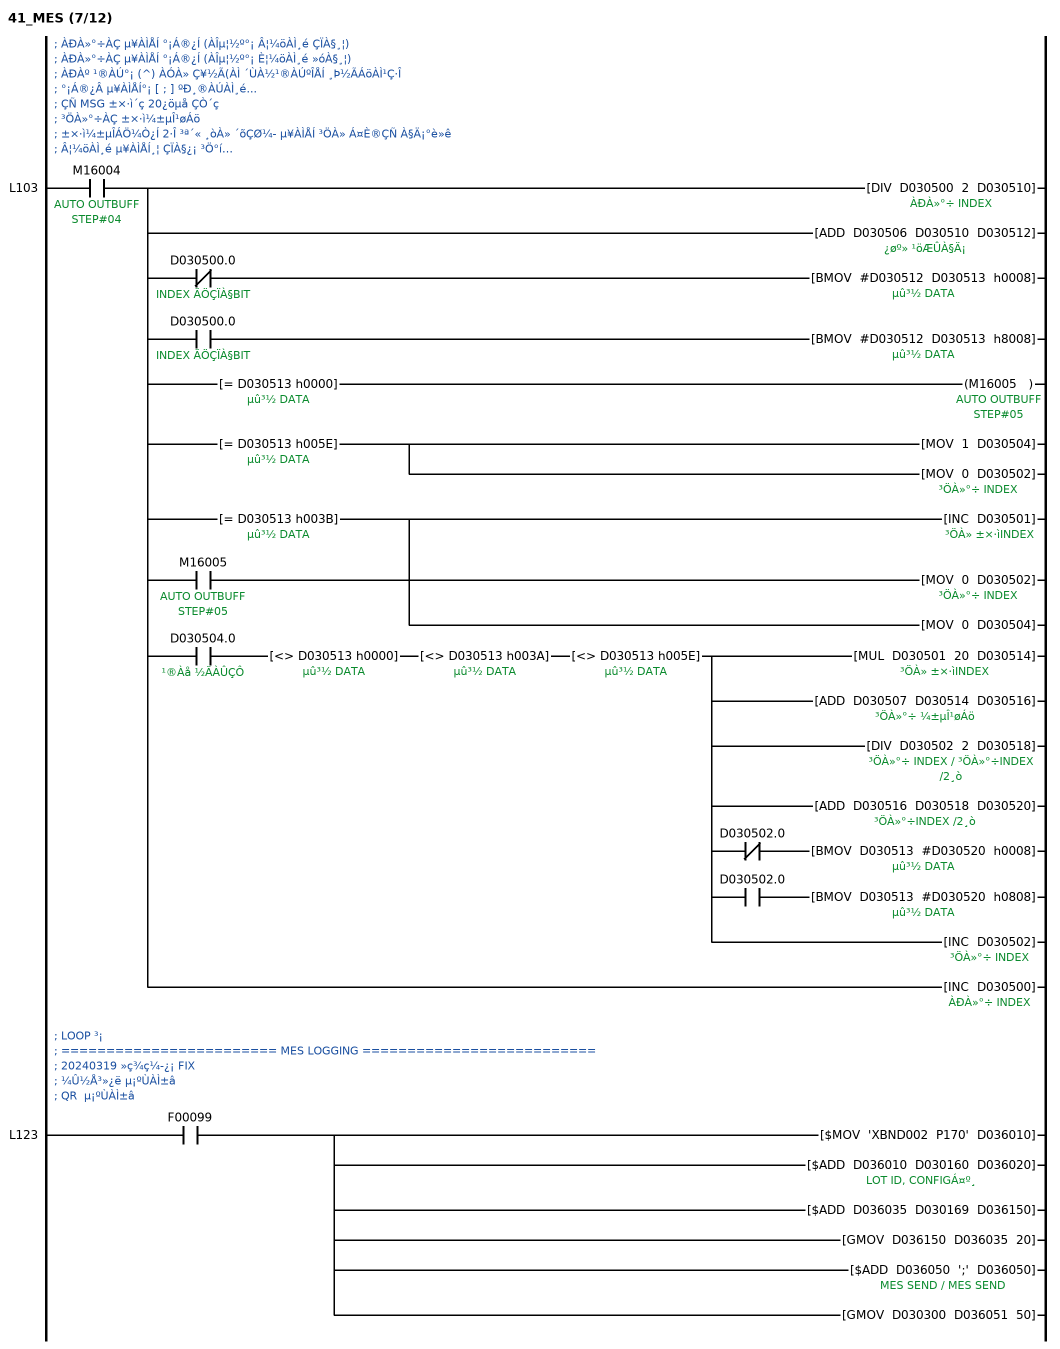
; L103
LOAD      M16004	// AUTO OUTBUFF STEP#04
DIV       D030500 2 D030510	// ÀÐÀ»°÷ INDEX
ADD       D030506 D030510 D030512	// ¿øº» ¹öÆÛÀ§Ä¡
MPUSH
AND NOT   D030500.0	// INDEX ÃÖÇÏÀ§BIT
BMOV      #D030512 D030513 h0008	// µû³½ DATA
MLOAD
AND       D030500.0	// INDEX ÃÖÇÏÀ§BIT
BMOV      #D030512 D030513 h8008	// µû³½ DATA
MLOAD
AND=      D030513 h0000	// µû³½ DATA
OUT       M16005	// AUTO OUTBUFF STEP#05
MLOAD
AND=      D030513 h005E	// µû³½ DATA
MOV       1 D030504
MOV       0 D030502	// ³ÖÀ»°÷ INDEX
MLOAD
LOAD=     D030513 h003B	// µû³½ DATA
OR        M16005	// AUTO OUTBUFF STEP#05
AND LOAD
INC       D030501	// ³ÖÀ» ±×·ìINDEX
MOV       0 D030502	// ³ÖÀ»°÷ INDEX
MOV       0 D030504
MLOAD
AND       D030504.0	// ¹®Àå ½ÃÀÛÇÔ
AND<>     D030513 h0000	// µû³½ DATA
AND<>     D030513 h003A	// µû³½ DATA
AND<>     D030513 h005E	// µû³½ DATA
MUL       D030501 20 D030514	// ³ÖÀ» ±×·ìINDEX
ADD       D030507 D030514 D030516	// ³ÖÀ»°÷ ¼±µÎ¹øÁö
DIV       D030502 2 D030518	// ³ÖÀ»°÷ INDEX / ³ÖÀ»°÷INDEX /2¸ò
ADD       D030516 D030518 D030520	// ³ÖÀ»°÷INDEX /2¸ò
MPUSH
AND NOT   D030502.0
BMOV      D030513 #D030520 h0008	// µû³½ DATA
MLOAD
AND       D030502.0
BMOV      D030513 #D030520 h0808	// µû³½ DATA
MPOP
INC       D030502	// ³ÖÀ»°÷ INDEX
MPOP
INC       D030500	// ÀÐÀ»°÷ INDEX
// output comment: ÀÐÀ»°÷ÀÇ µ¥ÀÌÅÍ °¡Á®¿Í (ÀÎµ¦½º°¡ Â¦¼öÀÌ¸é ÇÏÀ§¸¦)
// output comment: ÀÐÀ»°÷ÀÇ µ¥ÀÌÅÍ °¡Á®¿Í (ÀÎµ¦½º°¡ È¦¼öÀÌ¸é »óÀ§¸¦)
// output comment: ÀÐÀº ¹®ÀÚ°¡ (^) ÀÓÀ» Ç¥½Ã(ÀÌ ´ÙÀ½¹®ÀÚºÎÅÍ ¸Þ½ÃÁöÀÌ¹Ç·Î
// output comment: °¡Á®¿Â µ¥ÀÌÅÍ°¡ [ ; ] ºÐ¸®ÀÚÀÌ¸é...
// output comment: ÇÑ MSG ±×·ì´ç 20¿öµå ÇÒ´ç
// output comment: ³ÖÀ»°÷ÀÇ ±×·ì¼±µÎ¹øÁö
// output comment: ±×·ì¼±µÎÁÖ¼Ò¿Í 2·Î ³ª´« ¸òÀ» ´õÇØ¼­ µ¥ÀÌÅÍ ³ÖÀ» Á¤È®ÇÑ À§Ä¡°è»ê
// output comment: Â¦¼öÀÌ¸é µ¥ÀÌÅÍ¸¦ ÇÏÀ§¿¡ ³Ö°í,
// output comment: È¦¼öÀÌ¸é µ¥ÀÌÅÍ¸¦ »óÀ§¿¡ ³Ö¾î
// LOOP ³¡
// ======================== MES LOGGING ==========================
; L123
LOAD      F00099
$MOV      'XBND002  P170' D036010
$ADD      D036010 D030160 D036020	// LOT ID, CONFIGÁ¤º¸
$ADD      D036035 D030169 D036150
GMOV      D036150 D036035 20
$ADD      D036050 ';' D036050	// MES SEND / MES SEND
GMOV      D030300 D036051 50
// output comment: 20240319 »ç¾ç¼­¿¡ FIX
// output comment: ¼Û½Å³»¿ë µ¡ºÙÀÌ±â
// output comment: QR  µ¡ºÙÀÌ±â

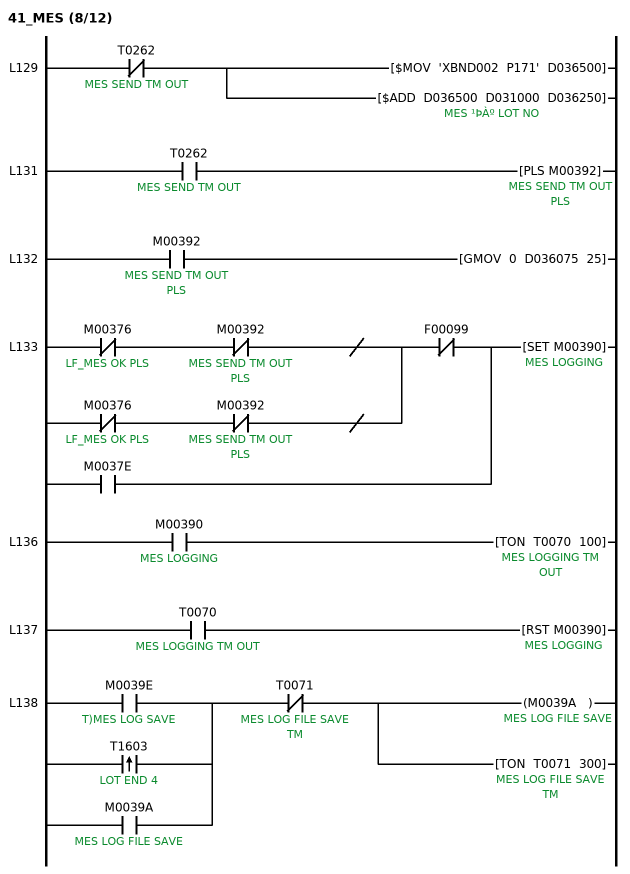
; L129
LOAD NOT  T0262	// MES SEND TM OUT
$MOV      'XBND002  P171' D036500
$ADD      D036500 D031000 D036250	// MES ¹ÞÀº LOT NO
; L131
LOAD      T0262	// MES SEND TM OUT
OUTP      M00392	// MES SEND TM OUT PLS
; L132
LOAD      M00392	// MES SEND TM OUT PLS
GMOV      0 D036075 25
; L133
LOAD NOT  M00376	// LF_MES OK PLS
AND NOT   M00392	// MES SEND TM OUT PLS
NOT
LOAD NOT  M00376	// LF_MES OK PLS
AND NOT   M00392	// MES SEND TM OUT PLS
NOT
OR LOAD
AND NOT   F00099
OR        M0037E
SET       M00390	// MES LOGGING
; L136
LOAD      M00390	// MES LOGGING
TON       T0070 100	// MES LOGGING TM OUT
; L137
LOAD      T0070	// MES LOGGING TM OUT
RST       M00390	// MES LOGGING
; L138
LOAD      M0039E	// T)MES LOG SAVE
ORP       T1603	// LOT END 4
OR        M0039A	// MES LOG FILE SAVE
AND NOT   T0071	// MES LOG FILE SAVE TM
OUT       M0039A	// MES LOG FILE SAVE
TON       T0071 300	// MES LOG FILE SAVE TM

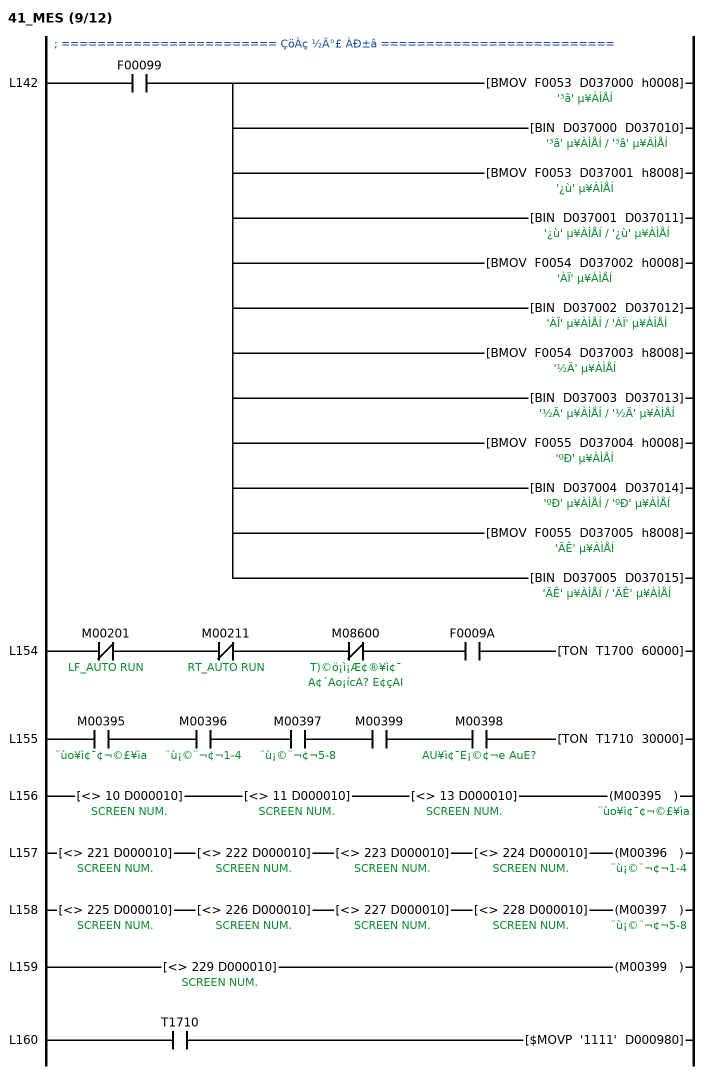
// ======================== ÇöÀç ½Ã°£ ÀÐ±â ==========================
; L142
LOAD      F00099
BMOV      F0053 D037000 h0008	// '³â' µ¥ÀÌÅÍ
BIN       D037000 D037010	// '³â' µ¥ÀÌÅÍ / '³â' µ¥ÀÌÅÍ
BMOV      F0053 D037001 h8008	// '¿ù' µ¥ÀÌÅÍ
BIN       D037001 D037011	// '¿ù' µ¥ÀÌÅÍ / '¿ù' µ¥ÀÌÅÍ
BMOV      F0054 D037002 h0008	// 'ÀÏ' µ¥ÀÌÅÍ
BIN       D037002 D037012	// 'ÀÏ' µ¥ÀÌÅÍ / 'ÀÏ' µ¥ÀÌÅÍ
BMOV      F0054 D037003 h8008	// '½Ã' µ¥ÀÌÅÍ
BIN       D037003 D037013	// '½Ã' µ¥ÀÌÅÍ / '½Ã' µ¥ÀÌÅÍ
BMOV      F0055 D037004 h0008	// 'ºÐ' µ¥ÀÌÅÍ
BIN       D037004 D037014	// 'ºÐ' µ¥ÀÌÅÍ / 'ºÐ' µ¥ÀÌÅÍ
BMOV      F0055 D037005 h8008	// 'ÃÊ' µ¥ÀÌÅÍ
BIN       D037005 D037015	// 'ÃÊ' µ¥ÀÌÅÍ / 'ÃÊ' µ¥ÀÌÅÍ
; L154
LOAD NOT  M00201	// LF_AUTO RUN
AND NOT   M00211	// RT_AUTO RUN
AND NOT   M08600	// T)©ö¡ì¡Æ¢®¥ì¢¯ A¢´Ao¡ícA? E¢çAI
AND       F0009A
TON       T1700 60000
; L155
LOAD      M00395	// ¨ùo¥ì¢¯¢¬©£¥ìa
AND       M00396	// ¨ù¡©¨¬¢¬1-4
AND       M00397	// ¨ù¡©¨¬¢¬5-8
AND       M00399
AND       M00398	// AU¥ì¢¯E¡©¢¬e AuE?
TON       T1710 30000
; L156
LOAD<>    10 D000010	// SCREEN NUM.
AND<>     11 D000010	// SCREEN NUM.
AND<>     13 D000010	// SCREEN NUM.
OUT       M00395	// ¨ùo¥ì¢¯¢¬©£¥ìa
; L157
LOAD<>    221 D000010	// SCREEN NUM.
AND<>     222 D000010	// SCREEN NUM.
AND<>     223 D000010	// SCREEN NUM.
AND<>     224 D000010	// SCREEN NUM.
OUT       M00396	// ¨ù¡©¨¬¢¬1-4
; L158
LOAD<>    225 D000010	// SCREEN NUM.
AND<>     226 D000010	// SCREEN NUM.
AND<>     227 D000010	// SCREEN NUM.
AND<>     228 D000010	// SCREEN NUM.
OUT       M00397	// ¨ù¡©¨¬¢¬5-8
; L159
LOAD<>    229 D000010	// SCREEN NUM.
OUT       M00399
; L160
LOAD      T1710
$MOVP     '1111' D000980

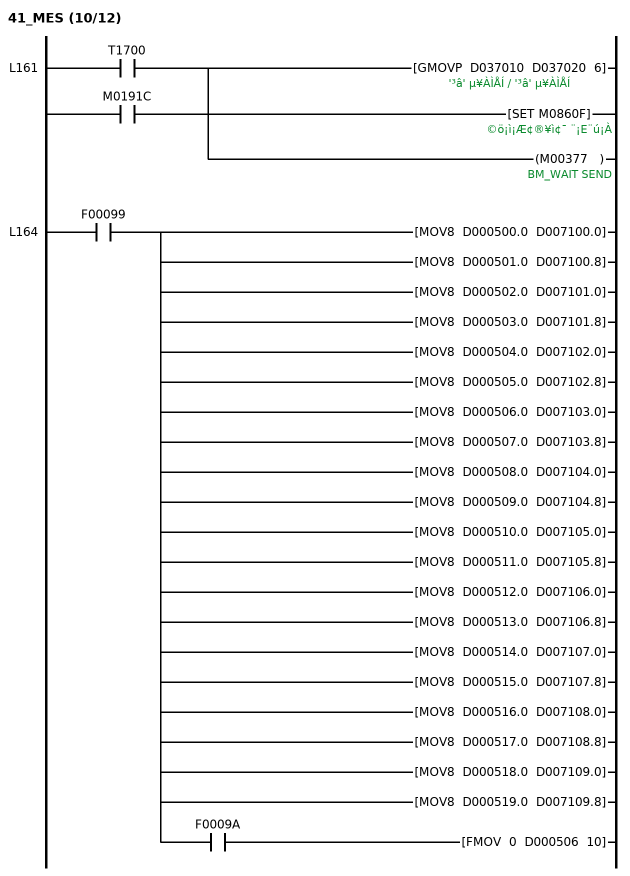
; L161
LOAD      T1700
OR        M0191C
GMOVP     D037010 D037020 6	// '³â' µ¥ÀÌÅÍ / '³â' µ¥ÀÌÅÍ
SET       M0860F	// ©ö¡ì¡Æ¢®¥ì¢¯ ¨¡E¨ú¡À
OUT       M00377	// BM_WAIT SEND
; L164
LOAD      F00099
MOV8      D000500.0 D007100.0
MOV8      D000501.0 D007100.8
MOV8      D000502.0 D007101.0
MOV8      D000503.0 D007101.8
MOV8      D000504.0 D007102.0
MOV8      D000505.0 D007102.8
MOV8      D000506.0 D007103.0
MOV8      D000507.0 D007103.8
MOV8      D000508.0 D007104.0
MOV8      D000509.0 D007104.8
MOV8      D000510.0 D007105.0
MOV8      D000511.0 D007105.8
MOV8      D000512.0 D007106.0
MOV8      D000513.0 D007106.8
MOV8      D000514.0 D007107.0
MOV8      D000515.0 D007107.8
MOV8      D000516.0 D007108.0
MOV8      D000517.0 D007108.8
MOV8      D000518.0 D007109.0
MOV8      D000519.0 D007109.8
AND       F0009A
FMOV      0 D000506 10

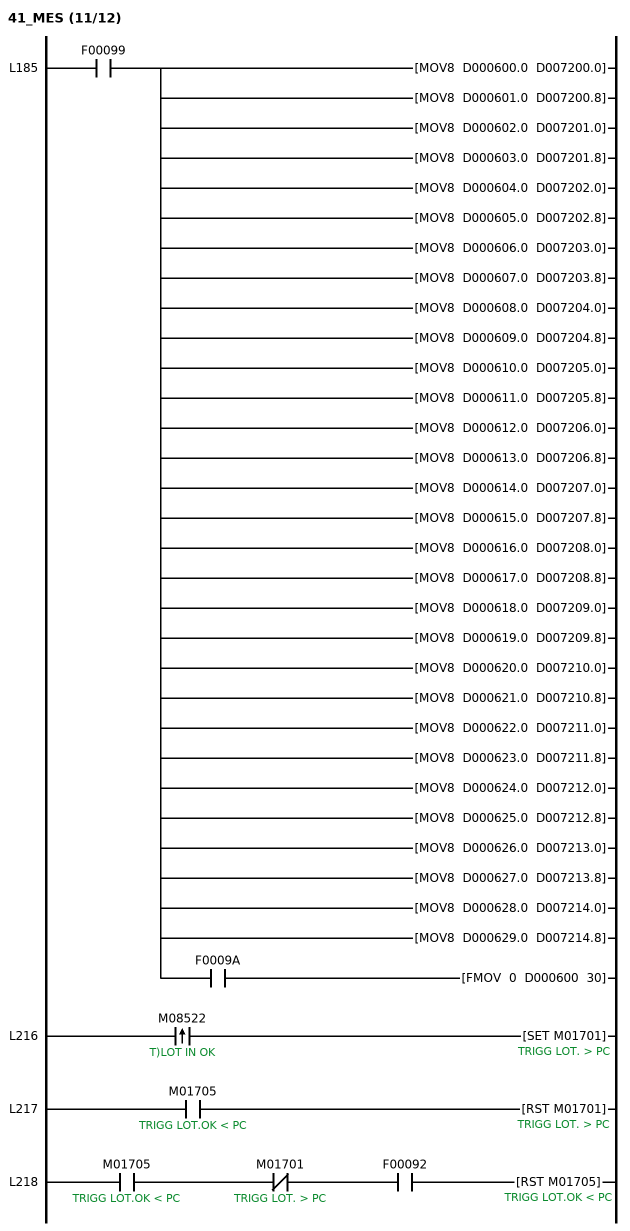
; L185
LOAD      F00099
MOV8      D000600.0 D007200.0
MOV8      D000601.0 D007200.8
MOV8      D000602.0 D007201.0
MOV8      D000603.0 D007201.8
MOV8      D000604.0 D007202.0
MOV8      D000605.0 D007202.8
MOV8      D000606.0 D007203.0
MOV8      D000607.0 D007203.8
MOV8      D000608.0 D007204.0
MOV8      D000609.0 D007204.8
MOV8      D000610.0 D007205.0
MOV8      D000611.0 D007205.8
MOV8      D000612.0 D007206.0
MOV8      D000613.0 D007206.8
MOV8      D000614.0 D007207.0
MOV8      D000615.0 D007207.8
MOV8      D000616.0 D007208.0
MOV8      D000617.0 D007208.8
MOV8      D000618.0 D007209.0
MOV8      D000619.0 D007209.8
MOV8      D000620.0 D007210.0
MOV8      D000621.0 D007210.8
MOV8      D000622.0 D007211.0
MOV8      D000623.0 D007211.8
MOV8      D000624.0 D007212.0
MOV8      D000625.0 D007212.8
MOV8      D000626.0 D007213.0
MOV8      D000627.0 D007213.8
MOV8      D000628.0 D007214.0
MOV8      D000629.0 D007214.8
AND       F0009A
FMOV      0 D000600 30
; L216
LOADP     M08522	// T)LOT IN OK
SET       M01701	// TRIGG LOT. > PC
; L217
LOAD      M01705	// TRIGG LOT.OK < PC
RST       M01701	// TRIGG LOT. > PC
; L218
LOAD      M01705	// TRIGG LOT.OK < PC
AND NOT   M01701	// TRIGG LOT. > PC
AND       F00092
RST       M01705	// TRIGG LOT.OK < PC

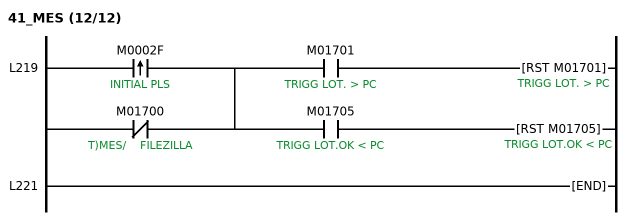
; L219
LOADP     M0002F	// INITIAL PLS
OR NOT    M01700	// T)MES/    FILEZILLA
MPUSH
AND       M01701	// TRIGG LOT. > PC
RST       M01701	// TRIGG LOT. > PC
MPOP
AND       M01705	// TRIGG LOT.OK < PC
RST       M01705	// TRIGG LOT.OK < PC
; L221
END

PROGRAM 51_MT_01_2_3_4 (task: ½ºÄµ ÇÁ·Î±×·¥)

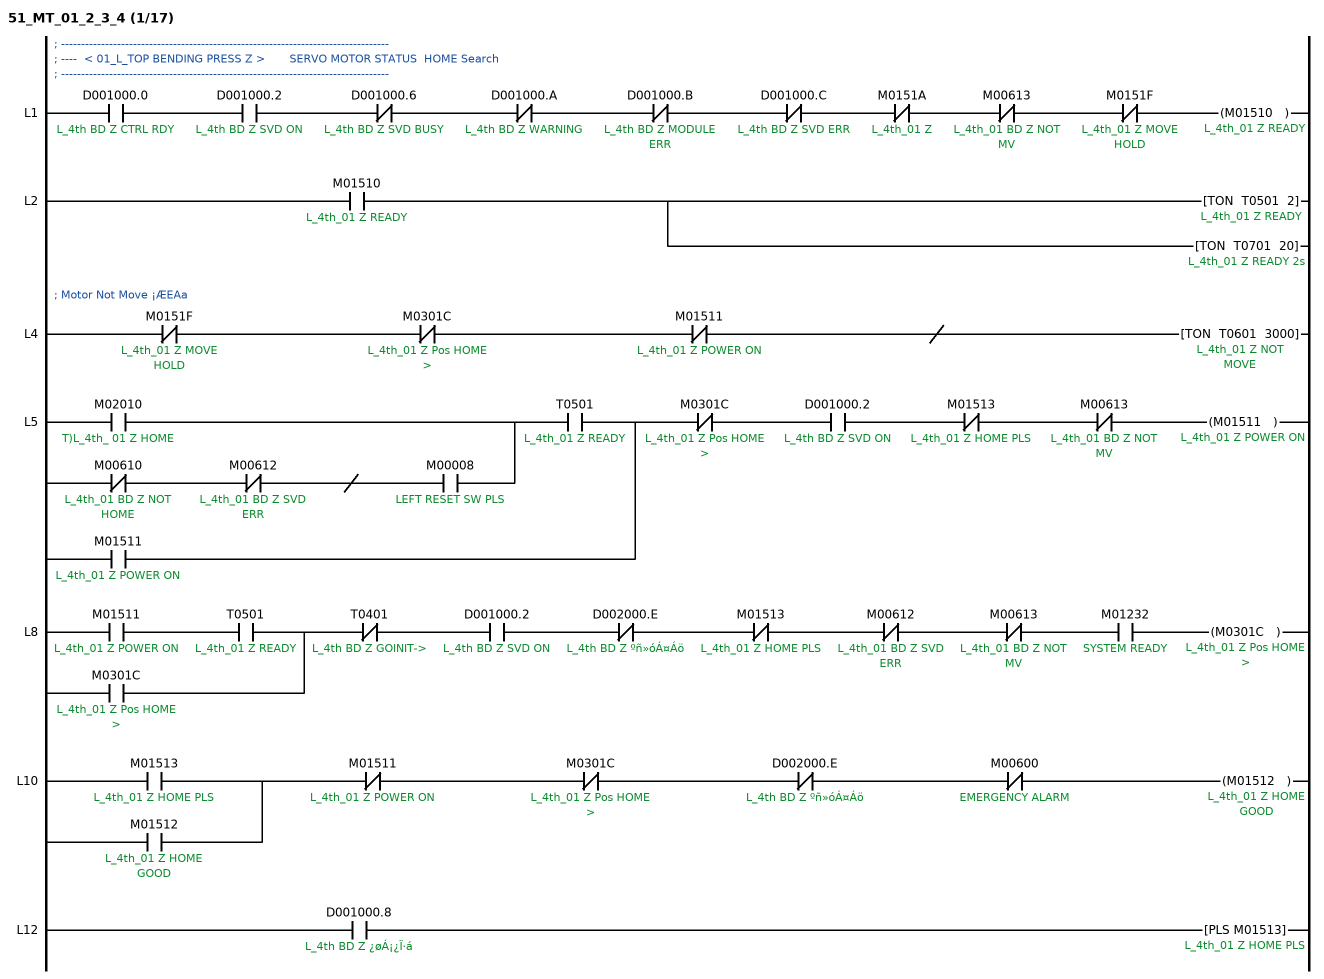
// ----------------------------------------------------------------------------------
// 
// ----  < 01_L_TOP BENDING PRESS Z >       SERVO MOTOR STATUS  HOME Search
// 
// ----------------------------------------------------------------------------------
; L1
LOAD      D001000.0	// L_4th BD Z CTRL RDY
AND       D001000.2	// L_4th BD Z SVD ON
AND NOT   D001000.6	// L_4th BD Z SVD BUSY
AND NOT   D001000.A	// L_4th BD Z WARNING
AND NOT   D001000.B	// L_4th BD Z MODULE ERR
AND NOT   D001000.C	// L_4th BD Z SVD ERR
AND NOT   M0151A	// L_4th_01 Z
AND NOT   M00613	// L_4th_01 BD Z NOT MV
AND NOT   M0151F	// L_4th_01 Z MOVE HOLD
OUT       M01510	// L_4th_01 Z READY
; L2
LOAD      M01510	// L_4th_01 Z READY
TON       T0501 2	// L_4th_01 Z READY
TON       T0701 20	// L_4th_01 Z READY 2s
; L4
LOAD NOT  M0151F	// L_4th_01 Z MOVE HOLD
AND NOT   M0301C	// L_4th_01 Z Pos HOME >
AND NOT   M01511	// L_4th_01 Z POWER ON
NOT
TON       T0601 3000	// L_4th_01 Z NOT MOVE
// output comment: Motor Not Move ¡ÆEAa
; L5
LOAD      M02010	// T)L_4th_ 01 Z HOME
LOAD NOT  M00610	// L_4th_01 BD Z NOT HOME
AND NOT   M00612	// L_4th_01 BD Z SVD ERR
NOT
AND       M00008	// LEFT RESET SW PLS
OR LOAD
AND       T0501	// L_4th_01 Z READY
OR        M01511	// L_4th_01 Z POWER ON
AND NOT   M0301C	// L_4th_01 Z Pos HOME >
AND       D001000.2	// L_4th BD Z SVD ON
AND NOT   M01513	// L_4th_01 Z HOME PLS
AND NOT   M00613	// L_4th_01 BD Z NOT MV
OUT       M01511	// L_4th_01 Z POWER ON
; L8
LOAD      M01511	// L_4th_01 Z POWER ON
AND       T0501	// L_4th_01 Z READY
OR        M0301C	// L_4th_01 Z Pos HOME >
AND NOT   T0401	// L_4th BD Z GOINIT->
AND       D001000.2	// L_4th BD Z SVD ON
AND NOT   D002000.E	// L_4th BD Z ºñ»óÁ¤Áö
AND NOT   M01513	// L_4th_01 Z HOME PLS
AND NOT   M00612	// L_4th_01 BD Z SVD ERR
AND NOT   M00613	// L_4th_01 BD Z NOT MV
AND       M01232	// SYSTEM READY
OUT       M0301C	// L_4th_01 Z Pos HOME >
; L10
LOAD      M01513	// L_4th_01 Z HOME PLS
OR        M01512	// L_4th_01 Z HOME GOOD
AND NOT   M01511	// L_4th_01 Z POWER ON
AND NOT   M0301C	// L_4th_01 Z Pos HOME >
AND NOT   D002000.E	// L_4th BD Z ºñ»óÁ¤Áö
AND NOT   M00600	// EMERGENCY ALARM
OUT       M01512	// L_4th_01 Z HOME GOOD
; L12
LOAD      D001000.8	// L_4th BD Z ¿øÁ¡¿Ï·á
OUTP      M01513	// L_4th_01 Z HOME PLS

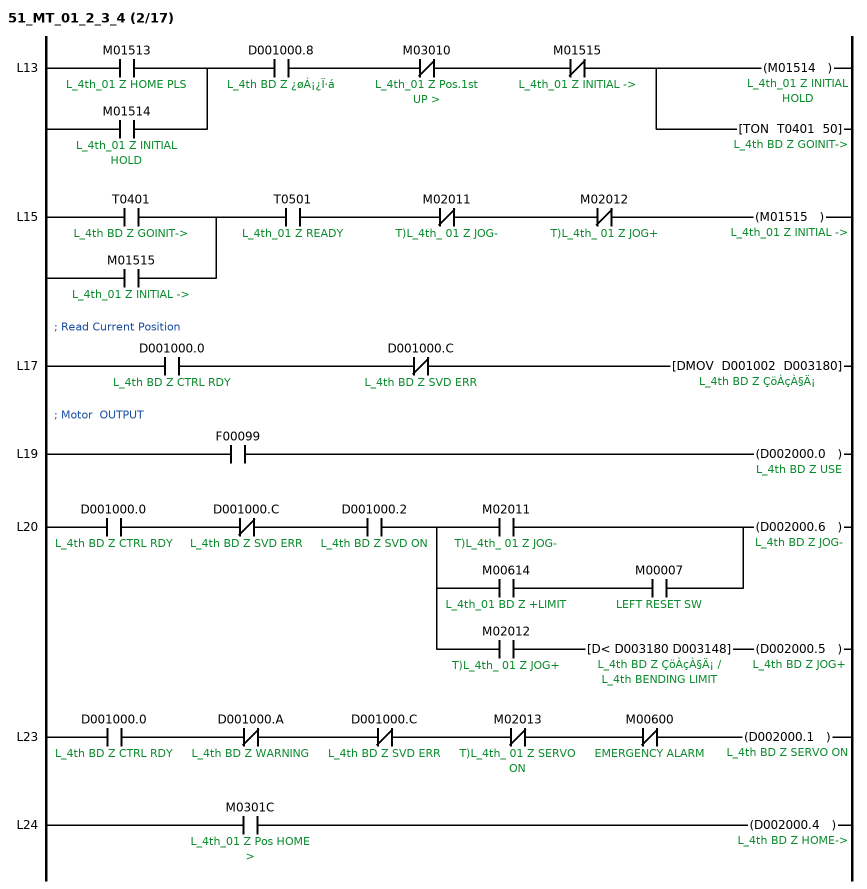
; L13
LOAD      M01513	// L_4th_01 Z HOME PLS
OR        M01514	// L_4th_01 Z INITIAL HOLD
AND       D001000.8	// L_4th BD Z ¿øÁ¡¿Ï·á
AND NOT   M03010	// L_4th_01 Z Pos.1st     UP >
AND NOT   M01515	// L_4th_01 Z INITIAL ->
OUT       M01514	// L_4th_01 Z INITIAL HOLD
TON       T0401 50	// L_4th BD Z GOINIT->
; L15
LOAD      T0401	// L_4th BD Z GOINIT->
OR        M01515	// L_4th_01 Z INITIAL ->
AND       T0501	// L_4th_01 Z READY
AND NOT   M02011	// T)L_4th_ 01 Z JOG-
AND NOT   M02012	// T)L_4th_ 01 Z JOG+
OUT       M01515	// L_4th_01 Z INITIAL ->
; L17
LOAD      D001000.0	// L_4th BD Z CTRL RDY
AND NOT   D001000.C	// L_4th BD Z SVD ERR
DMOV      D001002 D003180	// L_4th BD Z ÇöÀçÀ§Ä¡
// output comment: Read Current Position
//  Motor  OUTPUT
; L19
LOAD      F00099
OUT       D002000.0	// L_4th BD Z USE
; L20
LOAD      D001000.0	// L_4th BD Z CTRL RDY
AND NOT   D001000.C	// L_4th BD Z SVD ERR
AND       D001000.2	// L_4th BD Z SVD ON
MPUSH
LOAD      M02011	// T)L_4th_ 01 Z JOG-
LOAD      M00614	// L_4th_01 BD Z +LIMIT
AND       M00007	// LEFT RESET SW
OR LOAD
AND LOAD
OUT       D002000.6	// L_4th BD Z JOG-
MPOP
AND       M02012	// T)L_4th_ 01 Z JOG+
ANDD<     D003180 D003148	// L_4th BD Z ÇöÀçÀ§Ä¡ / L_4th BENDING LIMIT
OUT       D002000.5	// L_4th BD Z JOG+
; L23
LOAD      D001000.0	// L_4th BD Z CTRL RDY
AND NOT   D001000.A	// L_4th BD Z WARNING
AND NOT   D001000.C	// L_4th BD Z SVD ERR
AND NOT   M02013	// T)L_4th_ 01 Z SERVO ON
AND NOT   M00600	// EMERGENCY ALARM
OUT       D002000.1	// L_4th BD Z SERVO ON
; L24
LOAD      M0301C	// L_4th_01 Z Pos HOME >
OUT       D002000.4	// L_4th BD Z HOME->

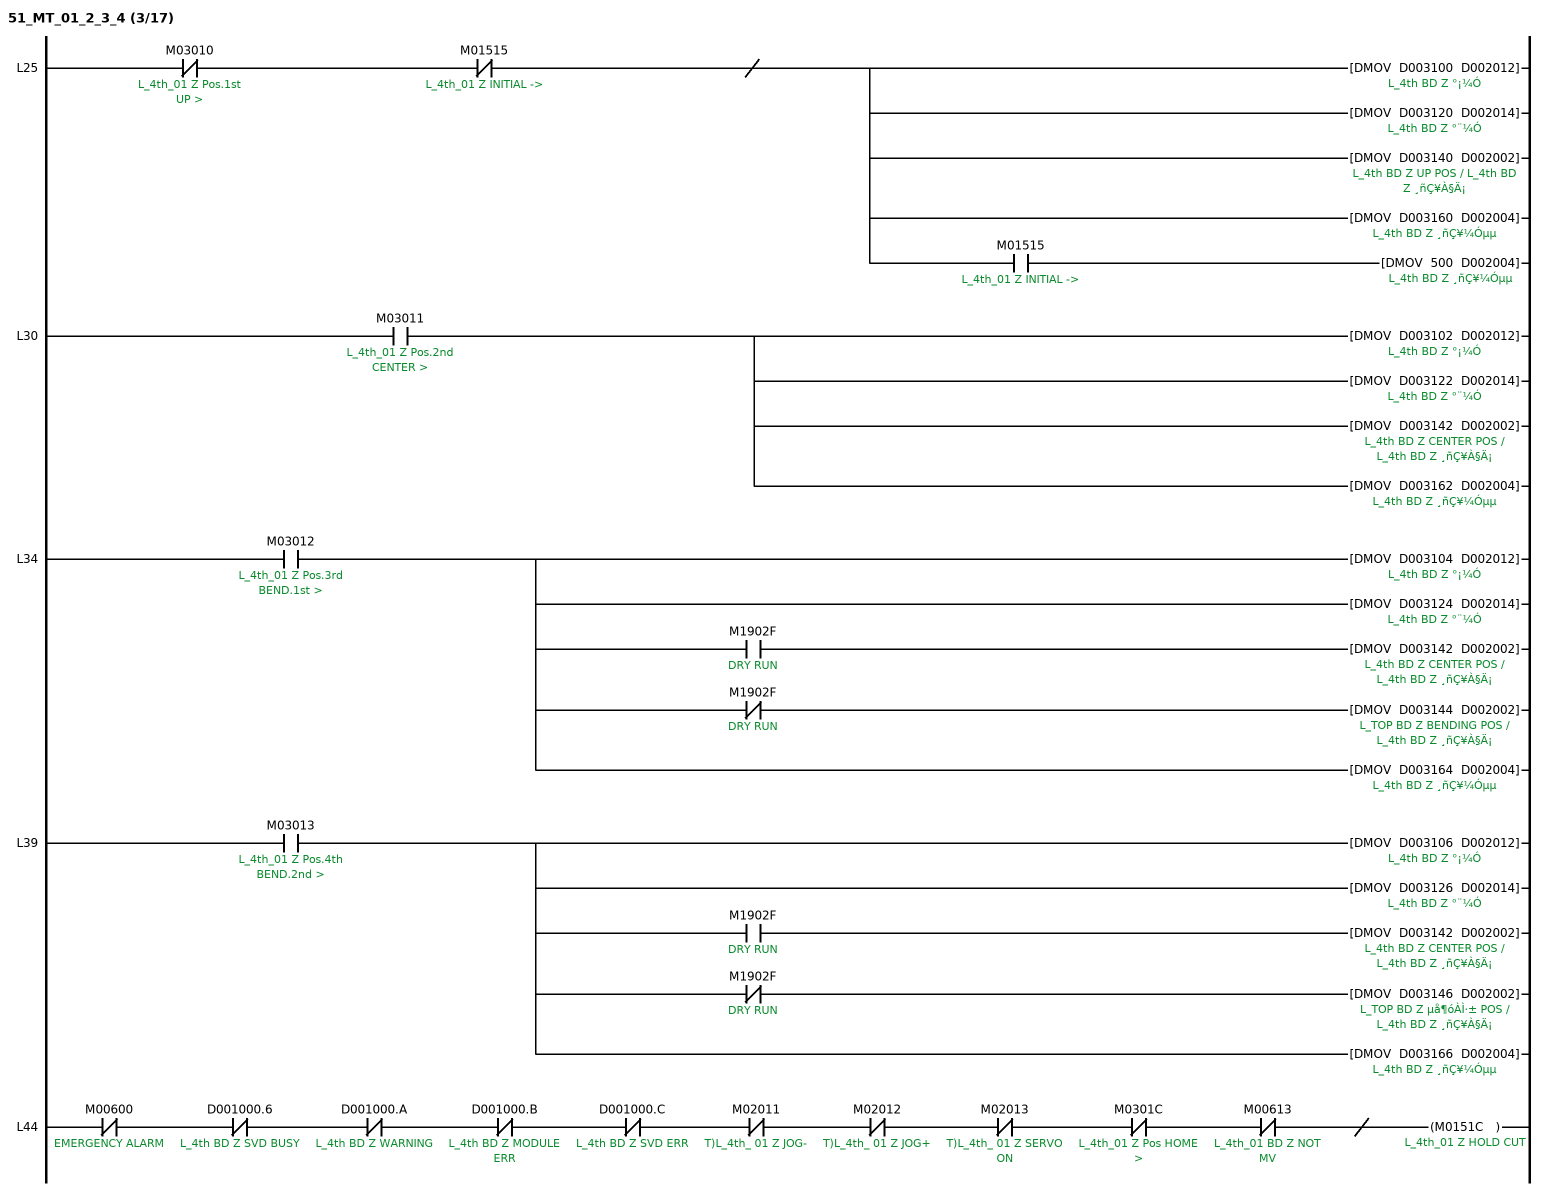
; L25
LOAD NOT  M03010	// L_4th_01 Z Pos.1st     UP >
AND NOT   M01515	// L_4th_01 Z INITIAL ->
NOT
DMOV      D003100 D002012	// L_4th BD Z °¡¼Ó
DMOV      D003120 D002014	// L_4th BD Z °¨¼Ó
DMOV      D003140 D002002	// L_4th BD Z UP POS / L_4th BD Z ¸ñÇ¥À§Ä¡
DMOV      D003160 D002004	// L_4th BD Z ¸ñÇ¥¼Óµµ
AND       M01515	// L_4th_01 Z INITIAL ->
DMOV      500 D002004	// L_4th BD Z ¸ñÇ¥¼Óµµ
; L30
LOAD      M03011	// L_4th_01 Z Pos.2nd CENTER >
DMOV      D003102 D002012	// L_4th BD Z °¡¼Ó
DMOV      D003122 D002014	// L_4th BD Z °¨¼Ó
DMOV      D003142 D002002	// L_4th BD Z CENTER POS / L_4th BD Z ¸ñÇ¥À§Ä¡
DMOV      D003162 D002004	// L_4th BD Z ¸ñÇ¥¼Óµµ
; L34
LOAD      M03012	// L_4th_01 Z Pos.3rd BEND.1st >
DMOV      D003104 D002012	// L_4th BD Z °¡¼Ó
DMOV      D003124 D002014	// L_4th BD Z °¨¼Ó
MPUSH
AND       M1902F	// DRY RUN
DMOV      D003142 D002002	// L_4th BD Z CENTER POS / L_4th BD Z ¸ñÇ¥À§Ä¡
MLOAD
AND NOT   M1902F	// DRY RUN
DMOV      D003144 D002002	// L_TOP BD Z BENDING POS / L_4th BD Z ¸ñÇ¥À§Ä¡
MPOP
DMOV      D003164 D002004	// L_4th BD Z ¸ñÇ¥¼Óµµ
; L39
LOAD      M03013	// L_4th_01 Z Pos.4th BEND.2nd >
DMOV      D003106 D002012	// L_4th BD Z °¡¼Ó
DMOV      D003126 D002014	// L_4th BD Z °¨¼Ó
MPUSH
AND       M1902F	// DRY RUN
DMOV      D003142 D002002	// L_4th BD Z CENTER POS / L_4th BD Z ¸ñÇ¥À§Ä¡
MLOAD
AND NOT   M1902F	// DRY RUN
DMOV      D003146 D002002	// L_TOP BD Z µå¶óÀÌ·± POS / L_4th BD Z ¸ñÇ¥À§Ä¡
MPOP
DMOV      D003166 D002004	// L_4th BD Z ¸ñÇ¥¼Óµµ
; L44
LOAD NOT  M00600	// EMERGENCY ALARM
AND NOT   D001000.6	// L_4th BD Z SVD BUSY
AND NOT   D001000.A	// L_4th BD Z WARNING
AND NOT   D001000.B	// L_4th BD Z MODULE ERR
AND NOT   D001000.C	// L_4th BD Z SVD ERR
AND NOT   M02011	// T)L_4th_ 01 Z JOG-
AND NOT   M02012	// T)L_4th_ 01 Z JOG+
AND NOT   M02013	// T)L_4th_ 01 Z SERVO ON
AND NOT   M0301C	// L_4th_01 Z Pos HOME >
AND NOT   M00613	// L_4th_01 BD Z NOT MV
NOT
OUT       M0151C	// L_4th_01 Z HOLD CUT

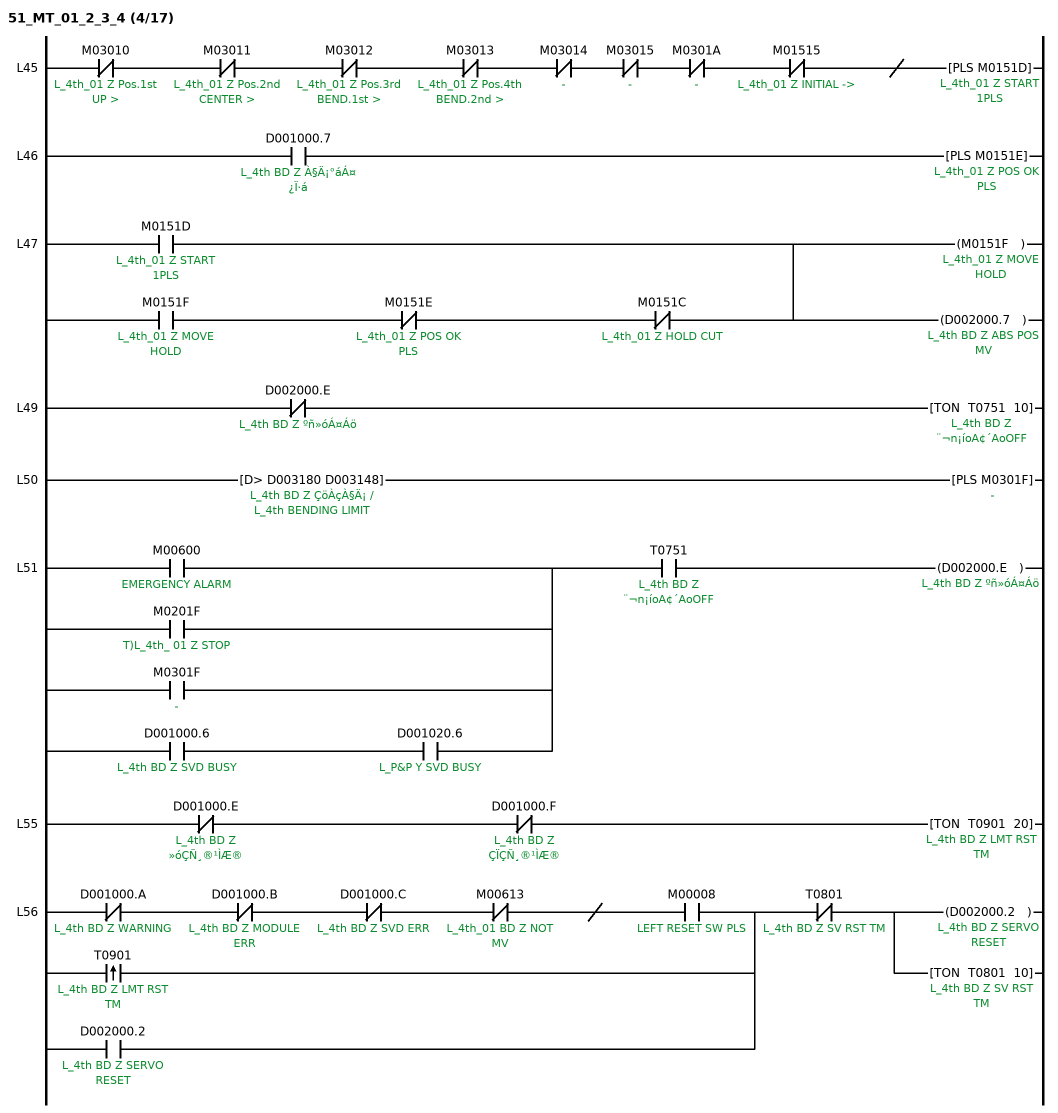
; L45
LOAD NOT  M03010	// L_4th_01 Z Pos.1st     UP >
AND NOT   M03011	// L_4th_01 Z Pos.2nd CENTER >
AND NOT   M03012	// L_4th_01 Z Pos.3rd BEND.1st >
AND NOT   M03013	// L_4th_01 Z Pos.4th BEND.2nd >
AND NOT   M03014	// -
AND NOT   M03015	// -
AND NOT   M0301A	// -
AND NOT   M01515	// L_4th_01 Z INITIAL ->
NOT
OUTP      M0151D	// L_4th_01 Z START 1PLS
; L46
LOAD      D001000.7	// L_4th BD Z À§Ä¡°áÁ¤ ¿Ï·á
OUTP      M0151E	// L_4th_01 Z POS OK PLS
; L47
LOAD      M0151D	// L_4th_01 Z START 1PLS
LOAD      M0151F	// L_4th_01 Z MOVE HOLD
AND NOT   M0151E	// L_4th_01 Z POS OK PLS
AND NOT   M0151C	// L_4th_01 Z HOLD CUT
OR LOAD
OUT       M0151F	// L_4th_01 Z MOVE HOLD
OUT       D002000.7	// L_4th BD Z ABS POS MV
; L49
LOAD NOT  D002000.E	// L_4th BD Z ºñ»óÁ¤Áö
TON       T0751 10	// L_4th BD Z ¨¬n¡íoA¢´AoOFF
; L50
LOADD>    D003180 D003148	// L_4th BD Z ÇöÀçÀ§Ä¡ / L_4th BENDING LIMIT
OUTP      M0301F	// -
; L51
LOAD      M00600	// EMERGENCY ALARM
OR        M0201F	// T)L_4th_ 01 Z STOP
OR        M0301F	// -
LOAD      D001000.6	// L_4th BD Z SVD BUSY
AND       D001020.6	// L_P&P Y SVD BUSY
OR LOAD
AND       T0751	// L_4th BD Z ¨¬n¡íoA¢´AoOFF
OUT       D002000.E	// L_4th BD Z ºñ»óÁ¤Áö
; L55
LOAD NOT  D001000.E	// L_4th BD Z »óÇÑ¸®¹ÌÆ®
AND NOT   D001000.F	// L_4th BD Z ÇÏÇÑ¸®¹ÌÆ®
TON       T0901 20	// L_4th BD Z LMT RST TM
; L56
LOAD NOT  D001000.A	// L_4th BD Z WARNING
AND NOT   D001000.B	// L_4th BD Z MODULE ERR
AND NOT   D001000.C	// L_4th BD Z SVD ERR
AND NOT   M00613	// L_4th_01 BD Z NOT MV
NOT
AND       M00008	// LEFT RESET SW PLS
ORP       T0901	// L_4th BD Z LMT RST TM
OR        D002000.2	// L_4th BD Z SERVO RESET
AND NOT   T0801	// L_4th BD Z SV RST TM
OUT       D002000.2	// L_4th BD Z SERVO RESET
TON       T0801 10	// L_4th BD Z SV RST TM

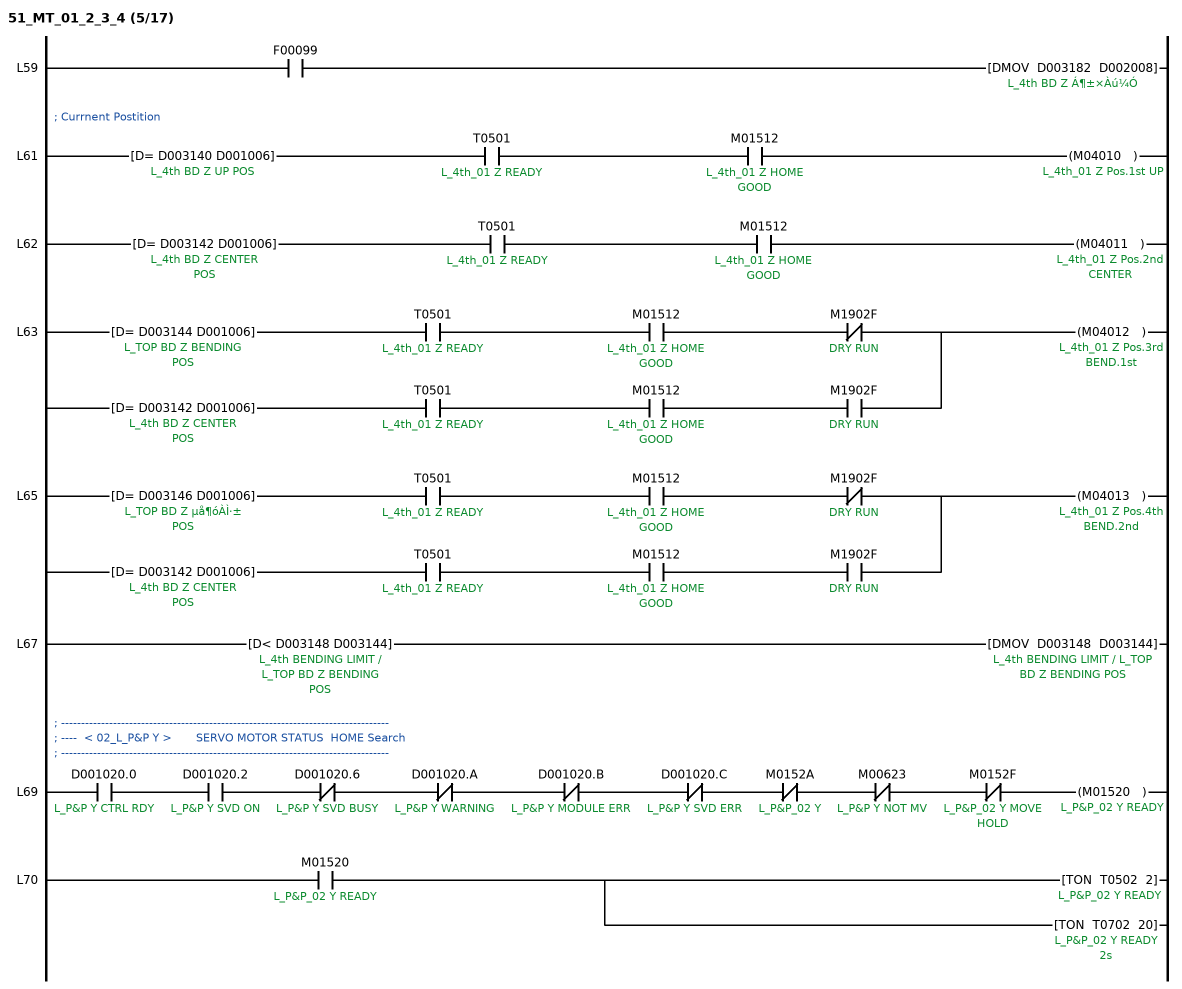
; L59
LOAD      F00099
DMOV      D003182 D002008	// L_4th BD Z Á¶±×Àú¼Ó
// Currnent Postition
; L61
LOADD=    D003140 D001006	// L_4th BD Z UP POS
AND       T0501	// L_4th_01 Z READY
AND       M01512	// L_4th_01 Z HOME GOOD
OUT       M04010	// L_4th_01 Z Pos.1st UP
; L62
LOADD=    D003142 D001006	// L_4th BD Z CENTER POS
AND       T0501	// L_4th_01 Z READY
AND       M01512	// L_4th_01 Z HOME GOOD
OUT       M04011	// L_4th_01 Z Pos.2nd CENTER
; L63
LOADD=    D003144 D001006	// L_TOP BD Z BENDING POS
AND       T0501	// L_4th_01 Z READY
AND       M01512	// L_4th_01 Z HOME GOOD
AND NOT   M1902F	// DRY RUN
LOADD=    D003142 D001006	// L_4th BD Z CENTER POS
AND       T0501	// L_4th_01 Z READY
AND       M01512	// L_4th_01 Z HOME GOOD
AND       M1902F	// DRY RUN
OR LOAD
OUT       M04012	// L_4th_01 Z Pos.3rd BEND.1st
; L65
LOADD=    D003146 D001006	// L_TOP BD Z µå¶óÀÌ·± POS
AND       T0501	// L_4th_01 Z READY
AND       M01512	// L_4th_01 Z HOME GOOD
AND NOT   M1902F	// DRY RUN
LOADD=    D003142 D001006	// L_4th BD Z CENTER POS
AND       T0501	// L_4th_01 Z READY
AND       M01512	// L_4th_01 Z HOME GOOD
AND       M1902F	// DRY RUN
OR LOAD
OUT       M04013	// L_4th_01 Z Pos.4th BEND.2nd
; L67
LOADD<    D003148 D003144	// L_4th BENDING LIMIT / L_TOP BD Z BENDING POS
DMOV      D003148 D003144	// L_4th BENDING LIMIT / L_TOP BD Z BENDING POS
// ----------------------------------------------------------------------------------
// 
// ----  < 02_L_P&P Y >       SERVO MOTOR STATUS  HOME Search
// 
// ----------------------------------------------------------------------------------
; L69
LOAD      D001020.0	// L_P&P Y CTRL RDY
AND       D001020.2	// L_P&P Y SVD ON
AND NOT   D001020.6	// L_P&P Y SVD BUSY
AND NOT   D001020.A	// L_P&P Y WARNING
AND NOT   D001020.B	// L_P&P Y MODULE ERR
AND NOT   D001020.C	// L_P&P Y SVD ERR
AND NOT   M0152A	// L_P&P_02 Y
AND NOT   M00623	// L_P&P Y NOT MV
AND NOT   M0152F	// L_P&P_02 Y MOVE HOLD
OUT       M01520	// L_P&P_02 Y READY
; L70
LOAD      M01520	// L_P&P_02 Y READY
TON       T0502 2	// L_P&P_02 Y READY
TON       T0702 20	// L_P&P_02 Y READY 2s

